KUKA KRL program: EPS_2_251806_MH42A_A_20260213065135.src

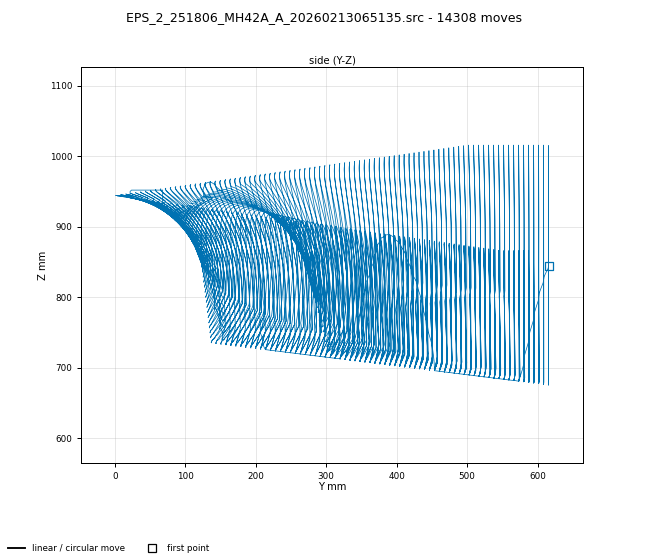
[picture p0: tool path of EPS_2_251806_MH42A_A_20260213065135.src, 14308 of 14310 moves have a stored position in this frame; points joined in program order, loops and branches not executed]
&ACCESS RVP
&REL 4
&COMMENT QRS 19112012
&PARAM EDITMASK = *
DEF PART()
EXT BAS (BAS_COMMAND :IN,REAL :IN )
INT I
BAS (#INITMOV,0 )

;KUKA QRS Post kuka4.cps  Date:22-06-2017 !

File_ID=3014

QRS_PRE_INIT()

;Init var - Until changes are made in qrs_pre_init
Outlet_Square_prg=0
Inlet_1_Square_prg=0
Inlet_2_Square_prg=0
Inlet_3_Square_prg=0
Inlet_4_Square_prg=0
Inlet_5_Square_prg=0

Outlet_1={X 0.000, Y 502.870, Z 915.500, B 0.000, E1 0.000 }
Inlet_1={X 0.000, Y 532.850, Z 495.500, B 0.000, E1 90.000 }
Inlet_2={X 0.000, Y 548.530, Z 275.500, B 0.000, E1 180.000 }
Outlet_1_type=201
Inlet_1_type=201
Inlet_2_type=201
;QRS#1=Sidecore dimensions
;QRS#2=200-8" PVC SDR 35
;QRS#3=200-8" PVC SDR 35
;QRS#4=200-8" PVC SDR 35
;QRS#5=
;QRS#6=
;QRS#7=
;QRS#8=
;QRS#9=12-08 PSX
;QRS#10=12-08 PSX
;QRS#11=12-08 PSX
;QRS#12=
;QRS#13=
;QRS#14=
;QRS#15=
;QRS#16=1220x127x1295 4,25'
;QRS#17=EPS Height
;QRS#18=1016
;QRS#19=*
;QRS#20= UPDATED VERSION 22-06-2017
;QRS#21=*
Outlet_Square=0100
Inlet_1_Square=0100
Inlet_2_Square=0100
Inlet_3_Square=0
Inlet_4_Square=0
Inlet_5_Square=0
Mill_Square=1
Outlet_Square_Prg=204
Inlet_1_Square_prg=204
Inlet_2_Square_prg=204

QRS_INIT()

$ADVANCE=5

; T1
PTP {E1 173.422,E2 173.422}
PTP {X 0,Y 615.492,A -85,B 0,C 180,E1 173.422,E2 173.422,E3 0,E4 0,E5 0,E6 0}
QRS_SPEED_INIT()
LIN {X 0,Y 615.492,Z 844.24,A -85,B 0,C 180,E1 173.422,E2 173.422,E3 0,E4 0,E5 0,E6 0} C_VEL
LIN {X 0,Y 615.497,Z 836.536,A -85,B 0,C 180,E1 172.455,E2 172.455} C_VEL
LIN {X 0,Y 615.498,Z 826.758,A -85,B 0,C 180,E1 171.463,E2 171.463} C_VEL
LIN {X 0,Y 615.497,Z 816.492,A -85,B 0,C 180,E1 170.636,E2 170.636} C_VEL
LIN {X 0,Y 615.468,Z 804.932,A -85,B 0,C 180,E1 169.888,E2 169.888} C_VEL
LIN {X 0,Y 615.49,Z 793.084,A -85,B 0,C 180,E1 169.293,E2 169.293} C_VEL
LIN {X 0,Y 615.491,Z 780.156,A -85,B 0,C 180,E1 168.807,E2 168.807} C_VEL
LIN {X 0,Y 615.484,Z 767.556,A -85,B 0,C 180,E1 168.473,E2 168.473} C_VEL
LIN {X 0,Y 615.469,Z 754.433,A -85,B 0,C 180,E1 168.264,E2 168.264} C_VEL
LIN {X 0,Y 615.494,Z 675.805,A -85,B 0,C 180,E1 167.344,E2 167.344} C_VEL
LIN {X 0,Y 615.486,Z 675.687,A -85,B 0,C 180,E1 164.774,E2 164.774} C_VEL
LIN {X 0,Y 615.473,Z 675.686,A -85,B 0,C 180,E1 162.043,E2 162.043} C_VEL
LIN {X 0,Y 615.491,Z 675.701,A -85,B 0,C 180,E1 159.269,E2 159.269} C_VEL
LIN {X 0,Y 615.483,Z 675.683,A -85,B 0,C 180,E1 156.443,E2 156.443} C_VEL
LIN {X 0,Y 615.479,Z 675.691,A -85,B 0,C 180,E1 153.555,E2 153.555} C_VEL
LIN {X 0,Y 615.487,Z 675.696,A -85,B 0,C 180,E1 151.342,E2 151.342} C_VEL
LIN {X 0,Y 615.478,Z 675.697,A -85,B 0,C 180,E1 148.917,E2 148.917} C_VEL
LIN {X 0,Y 615.465,Z 675.69,A -85,B 0,C 180,E1 146.471,E2 146.471} C_VEL
LIN {X 0,Y 615.468,Z 675.686,A -85,B 0,C 180,E1 144.171,E2 144.171} C_VEL
LIN {X 0,Y 615.479,Z 675.683,A -85,B 0,C 180,E1 141.931,E2 141.931} C_VEL
LIN {X 0,Y 615.486,Z 675.699,A -85,B 0,C 180,E1 138.908,E2 138.908} C_VEL
LIN {X 0,Y 615.474,Z 675.697,A -85,B 0,C 180,E1 136.754,E2 136.754} C_VEL
LIN {X 0,Y 615.447,Z 675.692,A -85,B 0,C 180,E1 134.155,E2 134.155} C_VEL
LIN {X 0,Y 615.487,Z 675.685,A -85,B 0,C 180,E1 131.476,E2 131.476} C_VEL
LIN {X 0,Y 615.493,Z 675.701,A -85,B 0,C 180,E1 128.906,E2 128.906} C_VEL
LIN {X 0,Y 615.45,Z 675.697,A -85,B 0,C 180,E1 126.43,E2 126.43} C_VEL
LIN {X 0,Y 615.431,Z 675.695,A -85,B 0,C 180,E1 124.028,E2 124.028} C_VEL
LIN {X 0,Y 615.432,Z 675.694,A -85,B 0,C 180,E1 121.691,E2 121.691} C_VEL
LIN {X 0,Y 615.443,Z 675.694,A -85,B 0,C 180,E1 119.411,E2 119.411} C_VEL
LIN {X 0,Y 615.456,Z 675.699,A -85,B 0,C 180,E1 116.448,E2 116.448} C_VEL
LIN {X 0,Y 615.415,Z 675.7,A -85,B 0,C 180,E1 113.992,E2 113.992} C_VEL
LIN {X 0,Y 615.425,Z 675.7,A -85,B 0,C 180,E1 112.142,E2 112.142} C_VEL
LIN {X 0,Y 615.418,Z 675.7,A -85,B 0,C 180,E1 110.038,E2 110.038} C_VEL
LIN {X 0,Y 615.418,Z 675.699,A -85,B 0,C 180,E1 107.962,E2 107.962} C_VEL
LIN {X 0,Y 615.422,Z 675.698,A -85,B 0,C 180,E1 105.91,E2 105.91} C_VEL
LIN {X 0,Y 615.427,Z 675.697,A -85,B 0,C 180,E1 103.879,E2 103.879} C_VEL
LIN {X 0,Y 615.489,Z 675.702,A -85,B 0,C 180,E1 102.576,E2 102.576} C_VEL
LIN {X 0,Y 615.42,Z 762.61,A -85,B 0,C 180,E1 101.532,E2 101.532} C_VEL
LIN {X 0,Y 615.425,Z 775.619,A -85,B 0,C 180,E1 101.24,E2 101.24} C_VEL
LIN {X 0,Y 615.46,Z 788.009,A -85,B 0,C 180,E1 100.828,E2 100.828} C_VEL
LIN {X 0,Y 615.489,Z 800.126,A -85,B 0,C 180,E1 100.281,E2 100.281} C_VEL
LIN {X 0,Y 615.483,Z 811.521,A -85,B 0,C 180,E1 99.617,E2 99.617} C_VEL
LIN {X 0,Y 615.498,Z 821.775,A -85,B 0,C 180,E1 98.871,E2 98.871} C_VEL
LIN {X 0,Y 615.498,Z 830.882,A -85,B 0,C 180,E1 98.044,E2 98.044} C_VEL
LIN {X 0,Y 615.497,Z 838.565,A -85,B 0,C 180,E1 97.219,E2 97.219} C_VEL
LIN {X 0,Y 615.497,Z 845.984,A -85,B 0,C 180,E1 96.231,E2 96.231} C_VEL
LIN {X 0,Y 615.497,Z 851.936,A -85,B 0,C 180,E1 95.245,E2 95.245} C_VEL
LIN {X 0,Y 615.493,Z 856.64,A -85,B 0,C 180,E1 94.26,E2 94.26} C_VEL
LIN {X 0,Y 615.494,Z 860.241,A -85,B 0,C 180,E1 93.277,E2 93.277} C_VEL
LIN {X 0,Y 615.496,Z 862.103,A -85,B 0,C 180,E1 92.622,E2 92.622} C_VEL
LIN {X 0,Y 615.497,Z 863.526,A -85,B 0,C 180,E1 91.967,E2 91.967} C_VEL
LIN {X 0,Y 615.496,Z 865.138,A -85,B 0,C 180,E1 90.659,E2 90.659} C_VEL
LIN {X 0,Y 615.495,Z 865.383,A -85,B 0,C 180,E1 90.004,E2 90.004} C_VEL
LIN {X 0,Y 615.495,Z 865.209,A -85,B 0,C 180,E1 89.35,E2 89.35} C_VEL
LIN {X 0,Y 615.497,Z 863.69,A -85,B 0,C 180,E1 88.041,E2 88.041} C_VEL
LIN {X 0,Y 615.498,Z 862.352,A -85,B 0,C 180,E1 87.387,E2 87.387} C_VEL
LIN {X 0,Y 615.496,Z 859.509,A -85,B 0,C 180,E1 86.404,E2 86.404} C_VEL
LIN {X 0,Y 615.499,Z 855.654,A -85,B 0,C 180,E1 85.42,E2 85.42} C_VEL
LIN {X 0,Y 615.498,Z 850.677,A -85,B 0,C 180,E1 84.435,E2 84.435} C_VEL
LIN {X 0,Y 615.488,Z 844.256,A -85,B 0,C 180,E1 83.424,E2 83.424} C_VEL
LIN {X 0,Y 615.497,Z 836.581,A -85,B 0,C 180,E1 82.46,E2 82.46} C_VEL
LIN {X 0,Y 615.498,Z 826.813,A -85,B 0,C 180,E1 81.469,E2 81.469} C_VEL
LIN {X 0,Y 615.497,Z 816.563,A -85,B 0,C 180,E1 80.641,E2 80.641} C_VEL
LIN {X 0,Y 615.486,Z 805.017,A -85,B 0,C 180,E1 79.894,E2 79.894} C_VEL
LIN {X 0,Y 615.485,Z 793.267,A -85,B 0,C 180,E1 79.301,E2 79.301} C_VEL
LIN {X 0,Y 615.438,Z 780.329,A -85,B 0,C 180,E1 78.811,E2 78.811} C_VEL
LIN {X 0,Y 615.427,Z 767.799,A -85,B 0,C 180,E1 78.477,E2 78.477} C_VEL
LIN {X 0,Y 615.431,Z 754.903,A -85,B 0,C 180,E1 78.269,E2 78.269} C_VEL
LIN {X 0,Y 615.491,Z 675.701,A -85,B 0,C 180,E1 77.329,E2 77.329} C_VEL
LIN {X 0,Y 615.444,Z 675.697,A -85,B 0,C 180,E1 74.778,E2 74.778} C_VEL
LIN {X 0,Y 615.445,Z 675.698,A -85,B 0,C 180,E1 72.734,E2 72.734} C_VEL
LIN {X 0,Y 615.441,Z 675.698,A -85,B 0,C 180,E1 70.667,E2 70.667} C_VEL
LIN {X 0,Y 615.441,Z 675.698,A -85,B 0,C 180,E1 68.573,E2 68.573} C_VEL
LIN {X 0,Y 615.435,Z 675.698,A -85,B 0,C 180,E1 66.448,E2 66.448} C_VEL
LIN {X 0,Y 615.429,Z 675.697,A -85,B 0,C 180,E1 64.288,E2 64.288} C_VEL
LIN {X 0,Y 615.424,Z 675.696,A -85,B 0,C 180,E1 62.089,E2 62.089} C_VEL
LIN {X 0,Y 615.422,Z 675.696,A -85,B 0,C 180,E1 59.844,E2 59.844} C_VEL
LIN {X 0,Y 615.428,Z 675.695,A -85,B 0,C 180,E1 57.547,E2 57.547} C_VEL
LIN {X 0,Y 615.45,Z 675.694,A -85,B 0,C 180,E1 55.191,E2 55.191} C_VEL
LIN {X 0,Y 615.49,Z 675.694,A -85,B 0,C 180,E1 52.766,E2 52.766} C_VEL
LIN {X 0,Y 615.43,Z 675.698,A -85,B 0,C 180,E1 49.918,E2 49.918} C_VEL
LIN {X 0,Y 615.42,Z 675.697,A -85,B 0,C 180,E1 47.651,E2 47.651} C_VEL
LIN {X 0,Y 615.439,Z 675.695,A -85,B 0,C 180,E1 44.937,E2 44.937} C_VEL
LIN {X 0,Y 615.474,Z 675.7,A -85,B 0,C 180,E1 42.09,E2 42.09} C_VEL
LIN {X 0,Y 615.44,Z 675.699,A -85,B 0,C 180,E1 39.754,E2 39.754} C_VEL
LIN {X 0,Y 615.411,Z 675.698,A -85,B 0,C 180,E1 37.248,E2 37.248} C_VEL
LIN {X 0,Y 615.428,Z 675.696,A -85,B 0,C 180,E1 34.706,E2 34.706} C_VEL
LIN {X 0,Y 615.458,Z 675.696,A -85,B 0,C 180,E1 32.341,E2 32.341} C_VEL
LIN {X 0,Y 615.434,Z 675.699,A -85,B 0,C 180,E1 29.409,E2 29.409} C_VEL
LIN {X 0,Y 615.414,Z 675.698,A -85,B 0,C 180,E1 27.049,E2 27.049} C_VEL
LIN {X 0,Y 615.414,Z 675.699,A -85,B 0,C 180,E1 24.995,E2 24.995} C_VEL
LIN {X 0,Y 615.407,Z 675.699,A -85,B 0,C 180,E1 22.848,E2 22.848} C_VEL
LIN {X 0,Y 615.409,Z 675.698,A -85,B 0,C 180,E1 20.56,E2 20.56} C_VEL
LIN {X 0,Y 615.444,Z 675.698,A -85,B 0,C 180,E1 17.958,E2 17.958} C_VEL
LIN {X 0,Y 615.462,Z 675.7,A -85,B 0,C 180,E1 15.227,E2 15.227} C_VEL
LIN {X 0,Y 615.407,Z 675.699,A -85,B 0,C 180,E1 12.532,E2 12.532} C_VEL
LIN {X 0,Y 615.408,Z 675.699,A -85,B 0,C 180,E1 10.528,E2 10.528} C_VEL
LIN {X 0,Y 615.411,Z 675.7,A -85,B 0,C 180,E1 8.538,E2 8.538} C_VEL
LIN {X 0,Y 615.415,Z 675.7,A -85,B 0,C 180,E1 6.558,E2 6.558} C_VEL
LIN {X 0,Y 615.422,Z 675.7,A -85,B 0,C 180,E1 4.585,E2 4.585} C_VEL
LIN {X 0,Y 615.43,Z 675.7,A -85,B 0,C 180,E1 2.618,E2 2.618} C_VEL
LIN {X 0,Y 615.401,Z 675.7,A -85,B 0,C 180,E1 0,E2 0} C_VEL
LIN {X 0,Y 615.431,Z 675.7,A -85,B 0,C 180,E1 -2.618,E2 -2.618} C_VEL
LIN {X 0,Y 615.479,Z 675.701,A -85,B 0,C 180,E1 -5.241,E2 -5.241} C_VEL
LIN {X 0,Y 615.418,Z 675.699,A -85,B 0,C 180,E1 -7.877,E2 -7.877} C_VEL
LIN {X 0,Y 615.425,Z 675.699,A -85,B 0,C 180,E1 -9.863,E2 -9.863} C_VEL
LIN {X 0,Y 615.431,Z 675.699,A -85,B 0,C 180,E1 -11.862,E2 -11.862} C_VEL
LIN {X 0,Y 615.431,Z 675.698,A -85,B 0,C 180,E1 -13.945,E2 -13.945} C_VEL
LIN {X 0,Y 615.408,Z 675.699,A -85,B 0,C 180,E1 -16.435,E2 -16.435} C_VEL
LIN {X 0,Y 615.408,Z 675.699,A -85,B 0,C 180,E1 -18.649,E2 -18.649} C_VEL
LIN {X 0,Y 615.466,Z 675.7,A -85,B 0,C 180,E1 -21.433,E2 -21.433} C_VEL
LIN {X 0,Y 615.434,Z 675.697,A -85,B 0,C 180,E1 -24.274,E2 -24.274} C_VEL
LIN {X 0,Y 615.425,Z 675.697,A -85,B 0,C 180,E1 -26.447,E2 -26.447} C_VEL
LIN {X 0,Y 615.417,Z 675.697,A -85,B 0,C 180,E1 -28.662,E2 -28.662} C_VEL
LIN {X 0,Y 615.412,Z 675.698,A -85,B 0,C 180,E1 -30.924,E2 -30.924} C_VEL
LIN {X 0,Y 615.436,Z 675.699,A -85,B 0,C 180,E1 -33.541,E2 -33.541} C_VEL
LIN {X 0,Y 615.466,Z 675.695,A -85,B 0,C 180,E1 -36.426,E2 -36.426} C_VEL
LIN {X 0,Y 615.425,Z 675.696,A -85,B 0,C 180,E1 -38.909,E2 -38.909} C_VEL
LIN {X 0,Y 615.419,Z 675.696,A -85,B 0,C 180,E1 -41.098,E2 -41.098} C_VEL
LIN {X 0,Y 615.418,Z 675.696,A -85,B 0,C 180,E1 -43.251,E2 -43.251} C_VEL
LIN {X 0,Y 615.434,Z 675.698,A -85,B 0,C 180,E1 -45.856,E2 -45.856} C_VEL
LIN {X 0,Y 615.497,Z 675.697,A -85,B 0,C 180,E1 -48.536,E2 -48.536} C_VEL
LIN {X 0,Y 615.442,Z 675.695,A -85,B 0,C 180,E1 -51.101,E2 -51.101} C_VEL
LIN {X 0,Y 615.421,Z 675.696,A -85,B 0,C 180,E1 -53.579,E2 -53.579} C_VEL
LIN {X 0,Y 615.469,Z 675.699,A -85,B 0,C 180,E1 -56.469,E2 -56.469} C_VEL
LIN {X 0,Y 615.475,Z 675.693,A -85,B 0,C 180,E1 -59.087,E2 -59.087} C_VEL
LIN {X 0,Y 615.437,Z 675.694,A -85,B 0,C 180,E1 -61.559,E2 -61.559} C_VEL
LIN {X 0,Y 615.423,Z 675.695,A -85,B 0,C 180,E1 -63.924,E2 -63.924} C_VEL
LIN {X 0,Y 615.422,Z 675.729,A -85,B 0,C 180,E1 -64.061,E2 -64.061} C_VEL
LIN {X 0,Y 615.468,Z 698.001,A -85,B 0,C 180,E1 -66.449,E2 -66.449} C_VEL
LIN {X 0,Y 615.49,Z 724.895,A -85,B 0,C 180,E1 -69.276,E2 -69.276} C_VEL
LIN {X 0,Y 615.484,Z 753.464,A -85,B 0,C 180,E1 -72.221,E2 -72.221} C_VEL
LIN {X 0,Y 615.437,Z 778.642,A -85,B 0,C 180,E1 -74.778,E2 -74.778} C_VEL
LIN {X 0,Y 615.451,Z 801.694,A -85,B 0,C 180,E1 -77.097,E2 -77.097} C_VEL
LIN {X 0,Y 615.434,Z 912.129,A -85,B 0,C 180,E1 -78.415,E2 -78.415} C_VEL
LIN {X 0,Y 615.441,Z 924.542,A -85,B 0,C 180,E1 -78.686,E2 -78.686} C_VEL
LIN {X 0,Y 615.479,Z 937.74,A -85,B 0,C 180,E1 -79.117,E2 -79.117} C_VEL
LIN {X 0,Y 615.492,Z 949.575,A -85,B 0,C 180,E1 -79.645,E2 -79.645} C_VEL
LIN {X 0,Y 615.483,Z 961.074,A -85,B 0,C 180,E1 -80.309,E2 -80.309} C_VEL
LIN {X 0,Y 615.499,Z 971.405,A -85,B 0,C 180,E1 -81.055,E2 -81.055} C_VEL
LIN {X 0,Y 615.497,Z 979.742,A -85,B 0,C 180,E1 -81.799,E2 -81.799} C_VEL
LIN {X 0,Y 615.497,Z 987.648,A -85,B 0,C 180,E1 -82.624,E2 -82.624} C_VEL
LIN {X 0,Y 615.491,Z 995.236,A -85,B 0,C 180,E1 -83.613,E2 -83.613} C_VEL
LIN {X 0,Y 615.498,Z 1002.23,A -85,B 0,C 180,E1 -84.764,E2 -84.764} C_VEL
LIN {X 0,Y 615.493,Z 1006.871,A -85,B 0,C 180,E1 -85.748,E2 -85.748} C_VEL
LIN {X 0,Y 615.494,Z 1010.413,A -85,B 0,C 180,E1 -86.732,E2 -86.732} C_VEL
LIN {X 0,Y 615.497,Z 1012.244,A -85,B 0,C 180,E1 -87.387,E2 -87.387} C_VEL
LIN {X 0,Y 615.497,Z 1013.616,A -85,B 0,C 180,E1 -88.041,E2 -88.041} C_VEL
LIN {X 0,Y 615.496,Z 1015.177,A -85,B 0,C 180,E1 -89.35,E2 -89.35} C_VEL
LIN {X 0,Y 615.494,Z 1015.389,A -85,B 0,C 180,E1 -90.004,E2 -90.004} C_VEL
LIN {X 0,Y 615.495,Z 1014.575,A -85,B 0,C 180,E1 -91.313,E2 -91.313} C_VEL
LIN {X 0,Y 615.497,Z 1013.601,A -85,B 0,C 180,E1 -91.967,E2 -91.967} C_VEL
LIN {X 0,Y 615.497,Z 1012.222,A -85,B 0,C 180,E1 -92.622,E2 -92.622} C_VEL
LIN {X 0,Y 615.495,Z 1009.336,A -85,B 0,C 180,E1 -93.605,E2 -93.605} C_VEL
LIN {X 0,Y 615.497,Z 1005.424,A -85,B 0,C 180,E1 -94.589,E2 -94.589} C_VEL
LIN {X 0,Y 615.499,Z 1000.383,A -85,B 0,C 180,E1 -95.574,E2 -95.574} C_VEL
LIN {X 0,Y 615.49,Z 993.913,A -85,B 0,C 180,E1 -96.578,E2 -96.578} C_VEL
LIN {X 0,Y 615.497,Z 986.099,A -85,B 0,C 180,E1 -97.549,E2 -97.549} C_VEL
LIN {X 0,Y 615.498,Z 976.214,A -85,B 0,C 180,E1 -98.54,E2 -98.54} C_VEL
LIN {X 0,Y 615.495,Z 965.813,A -85,B 0,C 180,E1 -99.368,E2 -99.368} C_VEL
LIN {X 0,Y 615.482,Z 955.513,A -85,B 0,C 180,E1 -100.032,E2 -100.032} C_VEL
LIN {X 0,Y 615.494,Z 944.086,A -85,B 0,C 180,E1 -100.618,E2 -100.618} C_VEL
LIN {X 0,Y 615.457,Z 932.311,A -85,B 0,C 180,E1 -101.079,E2 -101.079} C_VEL
LIN {X 0,Y 615.436,Z 919.092,A -85,B 0,C 180,E1 -101.448,E2 -101.448} C_VEL
LIN {X 0,Y 615.435,Z 905.652,A -85,B 0,C 180,E1 -101.677,E2 -101.677} C_VEL
LIN {X 0,Y 615.45,Z 801.605,A -85,B 0,C 180,E1 -102.912,E2 -102.912} C_VEL
LIN {X 0,Y 615.438,Z 776.876,A -85,B 0,C 180,E1 -105.4,E2 -105.4} C_VEL
LIN {X 0,Y 615.497,Z 751.695,A -85,B 0,C 180,E1 -107.96,E2 -107.96} C_VEL
LIN {X 0,Y 615.49,Z 724.806,A -85,B 0,C 180,E1 -110.734,E2 -110.734} C_VEL
LIN {X 0,Y 615.467,Z 697.911,A -85,B 0,C 180,E1 -113.56,E2 -113.56} C_VEL
LIN {X 0,Y 615.422,Z 675.85,A -85,B 0,C 180,E1 -115.926,E2 -115.926} C_VEL
LIN {X 0,Y 615.417,Z 675.698,A -85,B 0,C 180,E1 -117.921,E2 -117.921} C_VEL
LIN {X 0,Y 615.414,Z 675.698,A -85,B 0,C 180,E1 -120.167,E2 -120.167} C_VEL
LIN {X 0,Y 615.42,Z 675.699,A -85,B 0,C 180,E1 -122.464,E2 -122.464} C_VEL
LIN {X 0,Y 615.449,Z 675.7,A -85,B 0,C 180,E1 -124.82,E2 -124.82} C_VEL
LIN {X 0,Y 615.489,Z 675.699,A -85,B 0,C 180,E1 -127.244,E2 -127.244} C_VEL
LIN {X 0,Y 615.441,Z 675.696,A -85,B 0,C 180,E1 -129.756,E2 -129.756} C_VEL
LIN {X 0,Y 615.427,Z 675.695,A -85,B 0,C 180,E1 -132.074,E2 -132.074} C_VEL
LIN {X 0,Y 615.43,Z 675.695,A -85,B 0,C 180,E1 -134.157,E2 -134.157} C_VEL
LIN {X 0,Y 615.464,Z 675.698,A -85,B 0,C 180,E1 -136.957,E2 -136.957} C_VEL
LIN {X 0,Y 615.468,Z 675.688,A -85,B 0,C 180,E1 -139.915,E2 -139.915} C_VEL
LIN {X 0,Y 615.451,Z 675.695,A -85,B 0,C 180,E1 -142.755,E2 -142.755} C_VEL
LIN {X 0,Y 615.491,Z 675.701,A -85,B 0,C 180,E1 -145.301,E2 -145.301} C_VEL
LIN {X 0,Y 615.464,Z 675.687,A -85,B 0,C 180,E1 -148.313,E2 -148.313} C_VEL
LIN {X 0,Y 615.46,Z 675.689,A -85,B 0,C 180,E1 -150.592,E2 -150.592} C_VEL
LIN {X 0,Y 615.469,Z 675.694,A -85,B 0,C 180,E1 -152.96,E2 -152.96} C_VEL
LIN {X 0,Y 615.483,Z 675.691,A -85,B 0,C 180,E1 -155.728,E2 -155.728} C_VEL
LIN {X 0,Y 615.478,Z 675.684,A -85,B 0,C 180,E1 -158.568,E2 -158.568} C_VEL
LIN {X 0,Y 615.492,Z 675.702,A -85,B 0,C 180,E1 -161.396,E2 -161.396} C_VEL
LIN {X 0,Y 615.475,Z 675.686,A -85,B 0,C 180,E1 -164.094,E2 -164.094} C_VEL
LIN {X 0,Y 615.486,Z 675.685,A -85,B 0,C 180,E1 -166.799,E2 -166.799} C_VEL
LIN {X 0,Y 615.491,Z 675.702,A -85,B 0,C 180,E1 -167.428,E2 -167.428} C_VEL
LIN {X 0,Y 615.484,Z 761.644,A -85,B 0,C 180,E1 -168.452,E2 -168.452} C_VEL
LIN {X 0,Y 615.493,Z 774.222,A -85,B 0,C 180,E1 -168.724,E2 -168.724} C_VEL
LIN {X 0,Y 615.485,Z 786.478,A -85,B 0,C 180,E1 -169.116,E2 -169.116} C_VEL
LIN {X 0,Y 615.482,Z 798.567,A -85,B 0,C 180,E1 -169.639,E2 -169.639} C_VEL
LIN {X 0,Y 615.474,Z 810.307,A -85,B 0,C 180,E1 -170.304,E2 -170.304} C_VEL
LIN {X 0,Y 615.499,Z 820.768,A -85,B 0,C 180,E1 -171.05,E2 -171.05} C_VEL
LIN {X 0,Y 615.498,Z 829.231,A -85,B 0,C 180,E1 -171.794,E2 -171.794} C_VEL
LIN {X 0,Y 615.497,Z 837.209,A -85,B 0,C 180,E1 -172.62,E2 -172.62} C_VEL
LIN {X 0,Y 615.491,Z 844.9,A -85,B 0,C 180,E1 -173.608,E2 -173.608} C_VEL
LIN {X 0,Y 615.497,Z 851.958,A -85,B 0,C 180,E1 -174.759,E2 -174.759} C_VEL
LIN {X 0,Y 615.493,Z 856.658,A -85,B 0,C 180,E1 -175.744,E2 -175.744} C_VEL
LIN {X 0,Y 615.496,Z 860.254,A -85,B 0,C 180,E1 -176.727,E2 -176.727} C_VEL
LIN {X 0,Y 615.496,Z 862.115,A -85,B 0,C 180,E1 -177.382,E2 -177.382} C_VEL
LIN {X 0,Y 615.497,Z 863.534,A -85,B 0,C 180,E1 -178.037,E2 -178.037} C_VEL
LIN {X 0,Y 615.496,Z 865.142,A -85,B 0,C 180,E1 -179.346,E2 -179.346} C_VEL
LIN {X 0,Y 615.494,Z 865.384,A -85,B 0,C 180,E1 -180,E2 -180} C_VEL
LIN {X 0,Y 615.495,Z 865.206,A -85,B 0,C 180,E1 -180.654,E2 -180.654} C_VEL
LIN {X 0,Y 615.496,Z 863.683,A -85,B 0,C 180,E1 -181.963,E2 -181.963} C_VEL
LIN {X 0,Y 615.498,Z 862.341,A -85,B 0,C 180,E1 -182.618,E2 -182.618} C_VEL
LIN {X 0,Y 615.496,Z 859.494,A -85,B 0,C 180,E1 -183.601,E2 -183.601} C_VEL
LIN {X 0,Y 615.498,Z 855.634,A -85,B 0,C 180,E1 -184.585,E2 -184.585} C_VEL
LIN {X 0,Y 615.498,Z 850.651,A -85,B 0,C 180,E1 -185.57,E2 -185.57} C_VEL
LIN {X 0,Y 615.492,Z 844.24,A -85,B 0,C 180,E1 -186.578,E2 -186.578} C_VEL
LIN {X 0,Y 614.826,Z 841.059,A -85,B 0,C 180,E1 -187.027,E2 -187.027} C_VEL
LIN {X 0,Y 611.988,Z 835.485,A -85,B 0,C 180,E1 -187.745,E2 -187.745} C_VEL
LIN {X 0,Y 609.138,Z 829.212,A -85,B 0,C 180,E1 -188.426,E2 -188.426} C_VEL
LIN {X 0,Y 608.477,Z 824.972,A -85,B 0,C 180,E1 -188.816,E2 -188.816} C_VEL
LIN {X 0,Y 608.486,Z 814.391,A -85,B 0,C 180,E1 -189.641,E2 -189.641} C_VEL
LIN {X 0,Y 608.476,Z 803.599,A -85,B 0,C 180,E1 -190.313,E2 -190.313} C_VEL
LIN {X 0,Y 608.53,Z 791.933,A -85,B 0,C 180,E1 -190.885,E2 -190.885} C_VEL
LIN {X 0,Y 608.525,Z 778.959,A -85,B 0,C 180,E1 -191.365,E2 -191.365} C_VEL
LIN {X 0,Y 608.536,Z 766.652,A -85,B 0,C 180,E1 -191.681,E2 -191.681} C_VEL
LIN {X 0,Y 608.53,Z 752.744,A -85,B 0,C 180,E1 -191.893,E2 -191.893} C_VEL
LIN {X 0,Y 608.458,Z 676.695,A -85,B 0,C 180,E1 -192.805,E2 -192.805} C_VEL
LIN {X 0,Y 608.467,Z 676.686,A -85,B 0,C 180,E1 -195.406,E2 -195.406} C_VEL
LIN {X 0,Y 608.44,Z 676.691,A -85,B 0,C 180,E1 -198.172,E2 -198.172} C_VEL
LIN {X 0,Y 608.458,Z 676.693,A -85,B 0,C 180,E1 -200.982,E2 -200.982} C_VEL
LIN {X 0,Y 608.464,Z 676.685,A -85,B 0,C 180,E1 -203.845,E2 -203.845} C_VEL
LIN {X 0,Y 608.444,Z 676.688,A -85,B 0,C 180,E1 -206.036,E2 -206.036} C_VEL
LIN {X 0,Y 608.473,Z 676.691,A -85,B 0,C 180,E1 -208.618,E2 -208.618} C_VEL
LIN {X 0,Y 608.448,Z 676.691,A -85,B 0,C 180,E1 -211.318,E2 -211.318} C_VEL
LIN {X 0,Y 608.456,Z 676.687,A -85,B 0,C 180,E1 -213.731,E2 -213.731} C_VEL
LIN {X 0,Y 608.451,Z 676.687,A -85,B 0,C 180,E1 -216.092,E2 -216.092} C_VEL
LIN {X 0,Y 608.446,Z 676.692,A -85,B 0,C 180,E1 -218.59,E2 -218.59} C_VEL
LIN {X 0,Y 608.448,Z 676.692,A -85,B 0,C 180,E1 -221.339,E2 -221.339} C_VEL
LIN {X 0,Y 608.447,Z 676.688,A -85,B 0,C 180,E1 -223.872,E2 -223.872} C_VEL
LIN {X 0,Y 608.481,Z 676.688,A -85,B 0,C 180,E1 -226.69,E2 -226.69} C_VEL
LIN {X 0,Y 608.463,Z 676.692,A -85,B 0,C 180,E1 -228.822,E2 -228.822} C_VEL
LIN {X 0,Y 608.428,Z 676.696,A -85,B 0,C 180,E1 -231.406,E2 -231.406} C_VEL
LIN {X 0,Y 608.456,Z 676.697,A -85,B 0,C 180,E1 -233.083,E2 -233.083} C_VEL
LIN {X 0,Y 608.452,Z 676.692,A -85,B 0,C 180,E1 -235.527,E2 -235.527} C_VEL
LIN {X 0,Y 608.424,Z 676.691,A -85,B 0,C 180,E1 -237.9,E2 -237.9} C_VEL
LIN {X 0,Y 608.412,Z 676.692,A -85,B 0,C 180,E1 -240.215,E2 -240.215} C_VEL
LIN {X 0,Y 608.442,Z 676.691,A -85,B 0,C 180,E1 -242.8,E2 -242.8} C_VEL
LIN {X 0,Y 608.401,Z 676.695,A -85,B 0,C 180,E1 -245.864,E2 -245.864} C_VEL
LIN {X 0,Y 608.381,Z 676.696,A -85,B 0,C 180,E1 -248.302,E2 -248.302} C_VEL
LIN {X 0,Y 608.39,Z 676.695,A -85,B 0,C 180,E1 -250.424,E2 -250.424} C_VEL
LIN {X 0,Y 608.393,Z 676.694,A -85,B 0,C 180,E1 -252.518,E2 -252.518} C_VEL
LIN {X 0,Y 608.389,Z 676.695,A -85,B 0,C 180,E1 -254.588,E2 -254.588} C_VEL
LIN {X 0,Y 608.479,Z 676.872,A -85,B 0,C 180,E1 -257.298,E2 -257.298} C_VEL
LIN {X 0,Y 608.49,Z 762.745,A -85,B 0,C 180,E1 -258.335,E2 -258.335} C_VEL
LIN {X 0,Y 608.461,Z 776.507,A -85,B 0,C 180,E1 -258.651,E2 -258.651} C_VEL
LIN {X 0,Y 608.485,Z 787.939,A -85,B 0,C 180,E1 -259.038,E2 -259.038} C_VEL
LIN {X 0,Y 608.505,Z 800.289,A -85,B 0,C 180,E1 -259.6,E2 -259.6} C_VEL
LIN {X 0,Y 608.493,Z 811.722,A -85,B 0,C 180,E1 -260.271,E2 -260.271} C_VEL
LIN {X 0,Y 608.475,Z 822.026,A -85,B 0,C 180,E1 -261.026,E2 -261.026} C_VEL
LIN {X 0,Y 608.464,Z 831.203,A -85,B 0,C 180,E1 -261.862,E2 -261.862} C_VEL
LIN {X 0,Y 608.463,Z 838.934,A -85,B 0,C 180,E1 -262.697,E2 -262.697} C_VEL
LIN {X 0,Y 608.449,Z 846.41,A -85,B 0,C 180,E1 -263.696,E2 -263.696} C_VEL
LIN {X 0,Y 608.462,Z 852.413,A -85,B 0,C 180,E1 -264.694,E2 -264.694} C_VEL
LIN {X 0,Y 608.439,Z 857.161,A -85,B 0,C 180,E1 -265.69,E2 -265.69} C_VEL
LIN {X 0,Y 608.425,Z 860.799,A -85,B 0,C 180,E1 -266.685,E2 -266.685} C_VEL
LIN {X 0,Y 608.425,Z 862.679,A -85,B 0,C 180,E1 -267.348,E2 -267.348} C_VEL
LIN {X 0,Y 608.442,Z 864.119,A -85,B 0,C 180,E1 -268.01,E2 -268.01} C_VEL
LIN {X 0,Y 608.439,Z 865.749,A -85,B 0,C 180,E1 -269.334,E2 -269.334} C_VEL
LIN {X 0,Y 608.435,Z 865.994,A -85,B 0,C 180,E1 -269.996,E2 -269.996} C_VEL
LIN {X 0,Y 608.438,Z 865.818,A -85,B 0,C 180,E1 -270.657,E2 -270.657} C_VEL
LIN {X 0,Y 608.442,Z 864.284,A -85,B 0,C 180,E1 -271.981,E2 -271.981} C_VEL
LIN {X 0,Y 608.426,Z 862.929,A -85,B 0,C 180,E1 -272.644,E2 -272.644} C_VEL
LIN {X 0,Y 608.449,Z 860.057,A -85,B 0,C 180,E1 -273.638,E2 -273.638} C_VEL
LIN {X 0,Y 608.433,Z 856.164,A -85,B 0,C 180,E1 -274.633,E2 -274.633} C_VEL
LIN {X 0,Y 608.449,Z 851.139,A -85,B 0,C 180,E1 -275.63,E2 -275.63} C_VEL
LIN {X 0,Y 608.434,Z 844.828,A -85,B 0,C 180,E1 -276.628,E2 -276.628} C_VEL
LIN {X 0,Y 608.474,Z 836.917,A -85,B 0,C 180,E1 -277.628,E2 -277.628} C_VEL
LIN {X 0,Y 608.471,Z 827.084,A -85,B 0,C 180,E1 -278.631,E2 -278.631} C_VEL
LIN {X 0,Y 608.478,Z 816.787,A -85,B 0,C 180,E1 -279.468,E2 -279.468} C_VEL
LIN {X 0,Y 608.483,Z 805.19,A -85,B 0,C 180,E1 -280.224,E2 -280.224} C_VEL
LIN {X 0,Y 608.5,Z 793.1,A -85,B 0,C 180,E1 -280.836,E2 -280.836} C_VEL
LIN {X 0,Y 608.486,Z 780.417,A -85,B 0,C 180,E1 -281.318,E2 -281.318} C_VEL
LIN {X 0,Y 608.491,Z 767.871,A -85,B 0,C 180,E1 -281.656,E2 -281.656} C_VEL
LIN {X 0,Y 608.5,Z 754.992,A -85,B 0,C 180,E1 -281.867,E2 -281.867} C_VEL
LIN {X 0,Y 608.471,Z 676.694,A -85,B 0,C 180,E1 -282.799,E2 -282.799} C_VEL
LIN {X 0,Y 608.428,Z 676.691,A -85,B 0,C 180,E1 -285.401,E2 -285.401} C_VEL
LIN {X 0,Y 608.41,Z 676.693,A -85,B 0,C 180,E1 -287.472,E2 -287.472} C_VEL
LIN {X 0,Y 608.406,Z 676.694,A -85,B 0,C 180,E1 -289.566,E2 -289.566} C_VEL
LIN {X 0,Y 608.422,Z 676.691,A -85,B 0,C 180,E1 -291.687,E2 -291.687} C_VEL
LIN {X 0,Y 608.424,Z 676.69,A -85,B 0,C 180,E1 -294.14,E2 -294.14} C_VEL
LIN {X 0,Y 608.475,Z 676.694,A -85,B 0,C 180,E1 -297.206,E2 -297.206} C_VEL
LIN {X 0,Y 608.395,Z 676.694,A -85,B 0,C 180,E1 -299.959,E2 -299.959} C_VEL
LIN {X 0,Y 608.412,Z 676.692,A -85,B 0,C 180,E1 -302.09,E2 -302.09} C_VEL
LIN {X 0,Y 608.442,Z 676.691,A -85,B 0,C 180,E1 -304.904,E2 -304.904} C_VEL
LIN {X 0,Y 608.432,Z 676.695,A -85,B 0,C 180,E1 -307.74,E2 -307.74} C_VEL
LIN {X 0,Y 608.391,Z 676.695,A -85,B 0,C 180,E1 -310.322,E2 -310.322} C_VEL
LIN {X 0,Y 608.392,Z 676.695,A -85,B 0,C 180,E1 -312.327,E2 -312.327} C_VEL
LIN {X 0,Y 608.398,Z 676.693,A -85,B 0,C 180,E1 -314.791,E2 -314.791} C_VEL
LIN {X 0,Y 608.487,Z 676.692,A -85,B 0,C 180,E1 -317.652,E2 -317.652} C_VEL
LIN {X 0,Y 608.417,Z 676.691,A -85,B 0,C 180,E1 -320.556,E2 -320.556} C_VEL
LIN {X 0,Y 608.389,Z 676.695,A -85,B 0,C 180,E1 -323.08,E2 -323.08} C_VEL
LIN {X 0,Y 608.43,Z 676.693,A -85,B 0,C 180,E1 -325.528,E2 -325.528} C_VEL
LIN {X 0,Y 608.436,Z 676.697,A -85,B 0,C 180,E1 -327.904,E2 -327.904} C_VEL
LIN {X 0,Y 608.464,Z 676.694,A -85,B 0,C 180,E1 -330.22,E2 -330.22} C_VEL
LIN {X 0,Y 608.382,Z 676.695,A -85,B 0,C 180,E1 -333.222,E2 -333.222} C_VEL
LIN {X 0,Y 608.406,Z 676.696,A -85,B 0,C 180,E1 -334.697,E2 -334.697} C_VEL
LIN {X 0,Y 608.395,Z 676.696,A -85,B 0,C 180,E1 -336.874,E2 -336.874} C_VEL
LIN {X 0,Y 608.39,Z 676.694,A -85,B 0,C 180,E1 -339.318,E2 -339.318} C_VEL
LIN {X 0,Y 608.394,Z 676.695,A -85,B 0,C 180,E1 -341.826,E2 -341.826} C_VEL
LIN {X 0,Y 608.437,Z 676.699,A -85,B 0,C 180,E1 -344.593,E2 -344.593} C_VEL
LIN {X 0,Y 608.408,Z 676.693,A -85,B 0,C 180,E1 -347.322,E2 -347.322} C_VEL
LIN {X 0,Y 608.395,Z 676.695,A -85,B 0,C 180,E1 -349.349,E2 -349.349} C_VEL
LIN {X 0,Y 608.391,Z 676.696,A -85,B 0,C 180,E1 -351.363,E2 -351.363} C_VEL
LIN {X 0,Y 608.392,Z 676.696,A -85,B 0,C 180,E1 -353.366,E2 -353.366} C_VEL
LIN {X 0,Y 608.394,Z 676.696,A -85,B 0,C 180,E1 -355.362,E2 -355.362} C_VEL
LIN {X 0,Y 608.421,Z 676.694,A -85,B 0,C 180,E1 -357.352,E2 -357.352} C_VEL
LIN {X 0,Y 608.392,Z 676.694,A -85,B 0,C 180,E1 -360,E2 -360} C_VEL
LIN {X 0,Y 608.421,Z 676.694,A -85,B 0,C 180,E1 -362.648,E2 -362.648} C_VEL
LIN {X 0,Y 608.467,Z 676.693,A -85,B 0,C 180,E1 -365.302,E2 -365.302} C_VEL
LIN {X 0,Y 608.406,Z 676.693,A -85,B 0,C 180,E1 -367.968,E2 -367.968} C_VEL
LIN {X 0,Y 608.391,Z 676.695,A -85,B 0,C 180,E1 -369.978,E2 -369.978} C_VEL
LIN {X 0,Y 608.398,Z 676.695,A -85,B 0,C 180,E1 -372.001,E2 -372.001} C_VEL
LIN {X 0,Y 608.393,Z 676.695,A -85,B 0,C 180,E1 -374.039,E2 -374.039} C_VEL
LIN {X 0,Y 608.394,Z 676.694,A -85,B 0,C 180,E1 -376.534,E2 -376.534} C_VEL
LIN {X 0,Y 608.389,Z 676.695,A -85,B 0,C 180,E1 -378.872,E2 -378.872} C_VEL
LIN {X 0,Y 608.435,Z 676.699,A -85,B 0,C 180,E1 -381.693,E2 -381.693} C_VEL
LIN {X 0,Y 608.39,Z 676.694,A -85,B 0,C 180,E1 -384.574,E2 -384.574} C_VEL
LIN {X 0,Y 608.422,Z 676.697,A -85,B 0,C 180,E1 -386.037,E2 -386.037} C_VEL
LIN {X 0,Y 608.409,Z 676.692,A -85,B 0,C 180,E1 -389.023,E2 -389.023} C_VEL
LIN {X 0,Y 608.414,Z 676.693,A -85,B 0,C 180,E1 -391.32,E2 -391.32} C_VEL
LIN {X 0,Y 608.438,Z 676.695,A -85,B 0,C 180,E1 -393.744,E2 -393.744} C_VEL
LIN {X 0,Y 608.43,Z 676.701,A -85,B 0,C 180,E1 -396.094,E2 -396.094} C_VEL
LIN {X 0,Y 608.425,Z 676.693,A -85,B 0,C 180,E1 -398.591,E2 -398.591} C_VEL
LIN {X 0,Y 608.388,Z 676.694,A -85,B 0,C 180,E1 -401.182,E2 -401.182} C_VEL
LIN {X 0,Y 608.409,Z 676.692,A -85,B 0,C 180,E1 -403.313,E2 -403.313} C_VEL
LIN {X 0,Y 608.434,Z 676.696,A -85,B 0,C 180,E1 -406.137,E2 -406.137} C_VEL
LIN {X 0,Y 608.435,Z 676.693,A -85,B 0,C 180,E1 -408.831,E2 -408.831} C_VEL
LIN {X 0,Y 608.393,Z 676.694,A -85,B 0,C 180,E1 -411.415,E2 -411.415} C_VEL
LIN {X 0,Y 608.424,Z 676.693,A -85,B 0,C 180,E1 -413.091,E2 -413.091} C_VEL
LIN {X 0,Y 608.42,Z 676.69,A -85,B 0,C 180,E1 -415.536,E2 -415.536} C_VEL
LIN {X 0,Y 608.413,Z 676.692,A -85,B 0,C 180,E1 -417.91,E2 -417.91} C_VEL
LIN {X 0,Y 608.418,Z 676.693,A -85,B 0,C 180,E1 -420.225,E2 -420.225} C_VEL
LIN {X 0,Y 608.475,Z 676.695,A -85,B 0,C 180,E1 -422.794,E2 -422.794} C_VEL
LIN {X 0,Y 608.426,Z 676.779,A -85,B 0,C 180,E1 -423.855,E2 -423.855} C_VEL
LIN {X 0,Y 608.676,Z 680.188,A -85,B 0,C 180,E1 -424.24,E2 -424.24} C_VEL
LIN {X 0,Y 608.659,Z 706.573,A -85,B 0,C 180,E1 -427.089,E2 -427.089} C_VEL
LIN {X 0,Y 608.597,Z 731.618,A -85,B 0,C 180,E1 -429.737,E2 -429.737} C_VEL
LIN {X 0,Y 608.55,Z 756.832,A -85,B 0,C 180,E1 -432.359,E2 -432.359} C_VEL
LIN {X 0,Y 608.494,Z 782.045,A -85,B 0,C 180,E1 -434.943,E2 -434.943} C_VEL
LIN {X 0,Y 608.448,Z 801.916,A -85,B 0,C 180,E1 -436.957,E2 -436.957} C_VEL
LIN {X 0,Y 608.498,Z 912.233,A -85,B 0,C 180,E1 -438.281,E2 -438.281} C_VEL
LIN {X 0,Y 608.476,Z 925.405,A -85,B 0,C 180,E1 -438.576,E2 -438.576} C_VEL
LIN {X 0,Y 608.505,Z 937.727,A -85,B 0,C 180,E1 -438.986,E2 -438.986} C_VEL
LIN {X 0,Y 608.513,Z 949.734,A -85,B 0,C 180,E1 -439.525,E2 -439.525} C_VEL
LIN {X 0,Y 608.471,Z 961.275,A -85,B 0,C 180,E1 -440.196,E2 -440.196} C_VEL
LIN {X 0,Y 608.484,Z 971.658,A -85,B 0,C 180,E1 -440.951,E2 -440.951} C_VEL
LIN {X 0,Y 608.474,Z 980.051,A -85,B 0,C 180,E1 -441.704,E2 -441.704} C_VEL
LIN {X 0,Y 608.469,Z 988.003,A -85,B 0,C 180,E1 -442.539,E2 -442.539} C_VEL
LIN {X 0,Y 608.433,Z 995.318,A -85,B 0,C 180,E1 -443.489,E2 -443.489} C_VEL
LIN {X 0,Y 608.45,Z 1000.892,A -85,B 0,C 180,E1 -444.37,E2 -444.37} C_VEL
LIN {X 0,Y 608.432,Z 1005.97,A -85,B 0,C 180,E1 -445.367,E2 -445.367} C_VEL
LIN {X 0,Y 608.449,Z 1009.912,A -85,B 0,C 180,E1 -446.362,E2 -446.362} C_VEL
LIN {X 0,Y 608.425,Z 1012.821,A -85,B 0,C 180,E1 -447.356,E2 -447.356} C_VEL
LIN {X 0,Y 608.442,Z 1014.209,A -85,B 0,C 180,E1 -448.019,E2 -448.019} C_VEL
LIN {X 0,Y 608.438,Z 1015.787,A -85,B 0,C 180,E1 -449.343,E2 -449.343} C_VEL
LIN {X 0,Y 608.434,Z 1016,A -85,B 0,C 180,E1 -450.004,E2 -450.004} C_VEL
LIN {X 0,Y 608.448,Z 1015.179,A -85,B 0,C 180,E1 -451.328,E2 -451.328} C_VEL
LIN {X 0,Y 608.442,Z 1014.194,A -85,B 0,C 180,E1 -451.99,E2 -451.99} C_VEL
LIN {X 0,Y 608.425,Z 1012.798,A -85,B 0,C 180,E1 -452.652,E2 -452.652} C_VEL
LIN {X 0,Y 608.449,Z 1009.882,A -85,B 0,C 180,E1 -453.647,E2 -453.647} C_VEL
LIN {X 0,Y 608.432,Z 1005.932,A -85,B 0,C 180,E1 -454.642,E2 -454.642} C_VEL
LIN {X 0,Y 608.437,Z 999.852,A -85,B 0,C 180,E1 -455.805,E2 -455.805} C_VEL
LIN {X 0,Y 608.464,Z 993.206,A -85,B 0,C 180,E1 -456.803,E2 -456.803} C_VEL
LIN {X 0,Y 608.456,Z 984.954,A -85,B 0,C 180,E1 -457.804,E2 -457.804} C_VEL
LIN {X 0,Y 608.477,Z 974.554,A -85,B 0,C 180,E1 -458.807,E2 -458.807} C_VEL
LIN {X 0,Y 608.488,Z 963.691,A -85,B 0,C 180,E1 -459.645,E2 -459.645} C_VEL
LIN {X 0,Y 608.492,Z 952.703,A -85,B 0,C 180,E1 -460.317,E2 -460.317} C_VEL
LIN {X 0,Y 608.526,Z 940.912,A -85,B 0,C 180,E1 -460.884,E2 -460.884} C_VEL
LIN {X 0,Y 608.498,Z 928.767,A -85,B 0,C 180,E1 -461.327,E2 -461.327} C_VEL
LIN {X 0,Y 608.49,Z 916.315,A -85,B 0,C 180,E1 -461.644,E2 -461.644} C_VEL
LIN {X 0,Y 608.507,Z 900.423,A -85,B 0,C 180,E1 -461.876,E2 -461.876} C_VEL
LIN {X 0,Y 608.461,Z 802.051,A -85,B 0,C 180,E1 -463.041,E2 -463.041} C_VEL
LIN {X 0,Y 608.473,Z 778.594,A -85,B 0,C 180,E1 -465.409,E2 -465.409} C_VEL
LIN {X 0,Y 608.559,Z 753.381,A -85,B 0,C 180,E1 -467.998,E2 -467.998} C_VEL
LIN {X 0,Y 608.612,Z 726.679,A -85,B 0,C 180,E1 -470.782,E2 -470.782} C_VEL
LIN {X 0,Y 608.67,Z 699.592,A -85,B 0,C 180,E1 -473.659,E2 -473.659} C_VEL
LIN {X 0,Y 608.681,Z 679.592,A -85,B 0,C 180,E1 -475.825,E2 -475.825} C_VEL
LIN {X 0,Y 608.414,Z 676.694,A -85,B 0,C 180,E1 -476.178,E2 -476.178} C_VEL
LIN {X 0,Y 608.44,Z 676.692,A -85,B 0,C 180,E1 -478.614,E2 -478.614} C_VEL
LIN {X 0,Y 608.442,Z 676.696,A -85,B 0,C 180,E1 -481.321,E2 -481.321} C_VEL
LIN {X 0,Y 608.411,Z 676.694,A -85,B 0,C 180,E1 -483.726,E2 -483.726} C_VEL
LIN {X 0,Y 608.39,Z 676.695,A -85,B 0,C 180,E1 -486.099,E2 -486.099} C_VEL
LIN {X 0,Y 608.385,Z 676.695,A -85,B 0,C 180,E1 -488.23,E2 -488.23} C_VEL
LIN {X 0,Y 608.415,Z 676.692,A -85,B 0,C 180,E1 -490.325,E2 -490.325} C_VEL
LIN {X 0,Y 608.432,Z 676.696,A -85,B 0,C 180,E1 -492.964,E2 -492.964} C_VEL
LIN {X 0,Y 608.434,Z 676.692,A -85,B 0,C 180,E1 -495.741,E2 -495.741} C_VEL
LIN {X 0,Y 608.442,Z 676.689,A -85,B 0,C 180,E1 -497.937,E2 -497.937} C_VEL
LIN {X 0,Y 608.425,Z 676.693,A -85,B 0,C 180,E1 -500.71,E2 -500.71} C_VEL
LIN {X 0,Y 608.44,Z 676.696,A -85,B 0,C 180,E1 -503.084,E2 -503.084} C_VEL
LIN {X 0,Y 608.474,Z 676.691,A -85,B 0,C 180,E1 -505.531,E2 -505.531} C_VEL
LIN {X 0,Y 608.464,Z 676.687,A -85,B 0,C 180,E1 -507.905,E2 -507.905} C_VEL
LIN {X 0,Y 608.464,Z 676.685,A -85,B 0,C 180,E1 -510.22,E2 -510.22} C_VEL
LIN {X 0,Y 608.443,Z 676.691,A -85,B 0,C 180,E1 -512.801,E2 -512.801} C_VEL
LIN {X 0,Y 608.448,Z 676.697,A -85,B 0,C 180,E1 -515.429,E2 -515.429} C_VEL
LIN {X 0,Y 608.463,Z 676.686,A -85,B 0,C 180,E1 -518.308,E2 -518.308} C_VEL
LIN {X 0,Y 608.477,Z 676.693,A -85,B 0,C 180,E1 -521.284,E2 -521.284} C_VEL
LIN {X 0,Y 608.454,Z 676.69,A -85,B 0,C 180,E1 -523.906,E2 -523.906} C_VEL
LIN {X 0,Y 608.46,Z 676.687,A -85,B 0,C 180,E1 -526.643,E2 -526.643} C_VEL
LIN {X 0,Y 608.466,Z 676.694,A -85,B 0,C 180,E1 -527.291,E2 -527.291} C_VEL
LIN {X 0,Y 608.539,Z 761.772,A -85,B 0,C 180,E1 -528.319,E2 -528.319} C_VEL
LIN {X 0,Y 608.538,Z 775.113,A -85,B 0,C 180,E1 -528.614,E2 -528.614} C_VEL
LIN {X 0,Y 608.521,Z 788.484,A -85,B 0,C 180,E1 -529.059,E2 -529.059} C_VEL
LIN {X 0,Y 608.495,Z 800.36,A -85,B 0,C 180,E1 -529.603,E2 -529.603} C_VEL
LIN {X 0,Y 608.486,Z 811.782,A -85,B 0,C 180,E1 -530.275,E2 -530.275} C_VEL
LIN {X 0,Y 608.474,Z 822.08,A -85,B 0,C 180,E1 -531.029,E2 -531.029} C_VEL
LIN {X 0,Y 608.464,Z 831.243,A -85,B 0,C 180,E1 -531.866,E2 -531.866} C_VEL
LIN {X 0,Y 608.462,Z 838.965,A -85,B 0,C 180,E1 -532.701,E2 -532.701} C_VEL
LIN {X 0,Y 608.448,Z 846.435,A -85,B 0,C 180,E1 -533.7,E2 -533.7} C_VEL
LIN {X 0,Y 608.462,Z 852.433,A -85,B 0,C 180,E1 -534.698,E2 -534.698} C_VEL
LIN {X 0,Y 608.439,Z 857.177,A -85,B 0,C 180,E1 -535.694,E2 -535.694} C_VEL
LIN {X 0,Y 608.426,Z 860.811,A -85,B 0,C 180,E1 -536.689,E2 -536.689} C_VEL
LIN {X 0,Y 608.425,Z 862.691,A -85,B 0,C 180,E1 -537.352,E2 -537.352} C_VEL
LIN {X 0,Y 608.442,Z 864.127,A -85,B 0,C 180,E1 -538.014,E2 -538.014} C_VEL
LIN {X 0,Y 608.439,Z 865.752,A -85,B 0,C 180,E1 -539.338,E2 -539.338} C_VEL
LIN {X 0,Y 608.435,Z 865.995,A -85,B 0,C 180,E1 -540,E2 -540} C_VEL
LIN {X 0,Y 608.438,Z 865.815,A -85,B 0,C 180,E1 -540.662,E2 -540.662} C_VEL
LIN {X 0,Y 608.441,Z 864.276,A -85,B 0,C 180,E1 -541.986,E2 -541.986} C_VEL
LIN {X 0,Y 608.426,Z 862.917,A -85,B 0,C 180,E1 -542.648,E2 -542.648} C_VEL
LIN {X 0,Y 608.449,Z 860.04,A -85,B 0,C 180,E1 -543.642,E2 -543.642} C_VEL
LIN {X 0,Y 608.433,Z 856.141,A -85,B 0,C 180,E1 -544.638,E2 -544.638} C_VEL
LIN {X 0,Y 608.449,Z 851.111,A -85,B 0,C 180,E1 -545.634,E2 -545.634} C_VEL
LIN {X 0,Y 608.441,Z 844.794,A -85,B 0,C 180,E1 -546.633,E2 -546.633} C_VEL
LIN {X 0,Y 608.476,Z 836.877,A -85,B 0,C 180,E1 -547.633,E2 -547.633} C_VEL
LIN {X 0,Y 608.472,Z 827.029,A -85,B 0,C 180,E1 -548.636,E2 -548.636} C_VEL
LIN {X 0,Y 608.477,Z 824.972,A -85,B 0,C 180,E1 -548.816,E2 -548.816} C_VEL
LIN {X 0,Y 607.804,Z 820.637,A -85,B 0,C 180,E1 -549.187,E2 -549.187} C_VEL
LIN {X 0,Y 604.941,Z 813.394,A -85,B 0,C 180,E1 -549.766,E2 -549.766} C_VEL
LIN {X 0,Y 602.122,Z 805.767,A -85,B 0,C 180,E1 -550.298,E2 -550.298} C_VEL
LIN {X 0,Y 601.519,Z 800.688,A -85,B 0,C 180,E1 -550.591,E2 -550.591} C_VEL
LIN {X 0,Y 601.546,Z 788.829,A -85,B 0,C 180,E1 -551.146,E2 -551.146} C_VEL
LIN {X 0,Y 601.594,Z 776.057,A -85,B 0,C 180,E1 -551.583,E2 -551.583} C_VEL
LIN {X 0,Y 601.605,Z 763.197,A -85,B 0,C 180,E1 -551.882,E2 -551.882} C_VEL
LIN {X 0,Y 601.589,Z 725.864,A -85,B 0,C 180,E1 -552.353,E2 -552.353} C_VEL
LIN {X 0,Y 601.536,Z 678.231,A -85,B 0,C 180,E1 -552.925,E2 -552.925} C_VEL
LIN {X 0,Y 601.434,Z 677.568,A -85,B 0,C 180,E1 -552.957,E2 -552.957} C_VEL
LIN {X 0,Y 601.409,Z 677.565,A -85,B 0,C 180,E1 -555.592,E2 -555.592} C_VEL
LIN {X 0,Y 601.391,Z 677.567,A -85,B 0,C 180,E1 -557.689,E2 -557.689} C_VEL
LIN {X 0,Y 601.427,Z 677.569,A -85,B 0,C 180,E1 -560.522,E2 -560.522} C_VEL
LIN {X 0,Y 601.4,Z 677.567,A -85,B 0,C 180,E1 -563.411,E2 -563.411} C_VEL
LIN {X 0,Y 601.412,Z 677.564,A -85,B 0,C 180,E1 -565.865,E2 -565.865} C_VEL
LIN {X 0,Y 601.431,Z 677.568,A -85,B 0,C 180,E1 -568.627,E2 -568.627} C_VEL
LIN {X 0,Y 601.424,Z 677.565,A -85,B 0,C 180,E1 -571.453,E2 -571.453} C_VEL
LIN {X 0,Y 601.428,Z 677.562,A -85,B 0,C 180,E1 -574.119,E2 -574.119} C_VEL
LIN {X 0,Y 601.441,Z 677.564,A -85,B 0,C 180,E1 -577.381,E2 -577.381} C_VEL
LIN {X 0,Y 601.408,Z 677.564,A -85,B 0,C 180,E1 -579.996,E2 -579.996} C_VEL
LIN {X 0,Y 601.419,Z 677.568,A -85,B 0,C 180,E1 -582.67,E2 -582.67} C_VEL
LIN {X 0,Y 601.412,Z 677.567,A -85,B 0,C 180,E1 -585.478,E2 -585.478} C_VEL
LIN {X 0,Y 601.423,Z 677.564,A -85,B 0,C 180,E1 -588.407,E2 -588.407} C_VEL
LIN {X 0,Y 601.406,Z 677.571,A -85,B 0,C 180,E1 -590.871,E2 -590.871} C_VEL
LIN {X 0,Y 601.397,Z 677.572,A -85,B 0,C 180,E1 -593.414,E2 -593.414} C_VEL
LIN {X 0,Y 601.382,Z 677.568,A -85,B 0,C 180,E1 -596.072,E2 -596.072} C_VEL
LIN {X 0,Y 601.398,Z 677.567,A -85,B 0,C 180,E1 -598.549,E2 -598.549} C_VEL
LIN {X 0,Y 601.418,Z 677.572,A -85,B 0,C 180,E1 -601.37,E2 -601.37} C_VEL
LIN {X 0,Y 601.353,Z 677.571,A -85,B 0,C 180,E1 -604.145,E2 -604.145} C_VEL
LIN {X 0,Y 601.357,Z 677.572,A -85,B 0,C 180,E1 -606.584,E2 -606.584} C_VEL
LIN {X 0,Y 601.413,Z 677.572,A -85,B 0,C 180,E1 -609.474,E2 -609.474} C_VEL
LIN {X 0,Y 601.376,Z 677.575,A -85,B 0,C 180,E1 -611.603,E2 -611.603} C_VEL
LIN {X 0,Y 601.417,Z 677.569,A -85,B 0,C 180,E1 -613.709,E2 -613.709} C_VEL
LIN {X 0,Y 601.365,Z 677.57,A -85,B 0,C 180,E1 -616.479,E2 -616.479} C_VEL
LIN {X 0,Y 601.41,Z 677.571,A -85,B 0,C 180,E1 -617.147,E2 -617.147} C_VEL
LIN {X 0,Y 601.656,Z 682.281,A -85,B 0,C 180,E1 -617.216,E2 -617.216} C_VEL
LIN {X 0,Y 601.539,Z 762.773,A -85,B 0,C 180,E1 -618.198,E2 -618.198} C_VEL
LIN {X 0,Y 601.524,Z 776.533,A -85,B 0,C 180,E1 -618.519,E2 -618.519} C_VEL
LIN {X 0,Y 601.507,Z 788.977,A -85,B 0,C 180,E1 -618.95,E2 -618.95} C_VEL
LIN {X 0,Y 601.526,Z 800.287,A -85,B 0,C 180,E1 -619.478,E2 -619.478} C_VEL
LIN {X 0,Y 601.46,Z 811.717,A -85,B 0,C 180,E1 -620.157,E2 -620.157} C_VEL
LIN {X 0,Y 601.439,Z 822.019,A -85,B 0,C 180,E1 -620.92,E2 -620.92} C_VEL
LIN {X 0,Y 601.404,Z 831.221,A -85,B 0,C 180,E1 -621.766,E2 -621.766} C_VEL
LIN {X 0,Y 601.414,Z 838.943,A -85,B 0,C 180,E1 -622.611,E2 -622.611} C_VEL
LIN {X 0,Y 601.361,Z 846.334,A -85,B 0,C 180,E1 -623.609,E2 -623.609} C_VEL
LIN {X 0,Y 601.373,Z 852.42,A -85,B 0,C 180,E1 -624.631,E2 -624.631} C_VEL
LIN {X 0,Y 601.354,Z 857.166,A -85,B 0,C 180,E1 -625.639,E2 -625.639} C_VEL
LIN {X 0,Y 601.344,Z 860.803,A -85,B 0,C 180,E1 -626.646,E2 -626.646} C_VEL
LIN {X 0,Y 601.324,Z 862.679,A -85,B 0,C 180,E1 -627.316,E2 -627.316} C_VEL
LIN {X 0,Y 601.341,Z 864.113,A -85,B 0,C 180,E1 -627.986,E2 -627.986} C_VEL
LIN {X 0,Y 601.347,Z 865.127,A -85,B 0,C 180,E1 -628.656,E2 -628.656} C_VEL
LIN {X 0,Y 601.336,Z 865.986,A -85,B 0,C 180,E1 -629.996,E2 -629.996} C_VEL
LIN {X 0,Y 601.339,Z 865.818,A -85,B 0,C 180,E1 -630.665,E2 -630.665} C_VEL
LIN {X 0,Y 601.341,Z 864.282,A -85,B 0,C 180,E1 -632.005,E2 -632.005} C_VEL
LIN {X 0,Y 601.326,Z 862.928,A -85,B 0,C 180,E1 -632.675,E2 -632.675} C_VEL
LIN {X 0,Y 601.367,Z 860.057,A -85,B 0,C 180,E1 -633.681,E2 -633.681} C_VEL
LIN {X 0,Y 601.337,Z 856.164,A -85,B 0,C 180,E1 -634.688,E2 -634.688} C_VEL
LIN {X 0,Y 601.372,Z 851.14,A -85,B 0,C 180,E1 -635.696,E2 -635.696} C_VEL
LIN {X 0,Y 601.376,Z 844.821,A -85,B 0,C 180,E1 -636.706,E2 -636.706} C_VEL
LIN {X 0,Y 601.394,Z 836.901,A -85,B 0,C 180,E1 -637.718,E2 -637.718} C_VEL
LIN {X 0,Y 601.421,Z 828.818,A -85,B 0,C 180,E1 -638.563,E2 -638.563} C_VEL
LIN {X 0,Y 601.451,Z 819.019,A -85,B 0,C 180,E1 -639.41,E2 -639.41} C_VEL
LIN {X 0,Y 601.486,Z 808.011,A -85,B 0,C 180,E1 -640.174,E2 -640.174} C_VEL
LIN {X 0,Y 601.528,Z 795.677,A -85,B 0,C 180,E1 -640.844,E2 -640.844} C_VEL
LIN {X 0,Y 601.498,Z 783.842,A -85,B 0,C 180,E1 -641.335,E2 -641.335} C_VEL
LIN {X 0,Y 601.518,Z 771.47,A -85,B 0,C 180,E1 -641.707,E2 -641.707} C_VEL
LIN {X 0,Y 601.549,Z 758.138,A -85,B 0,C 180,E1 -641.963,E2 -641.963} C_VEL
LIN {X 0,Y 601.581,Z 678.471,A -85,B 0,C 180,E1 -642.921,E2 -642.921} C_VEL
LIN {X 0,Y 601.412,Z 677.571,A -85,B 0,C 180,E1 -642.952,E2 -642.952} C_VEL
LIN {X 0,Y 601.373,Z 677.569,A -85,B 0,C 180,E1 -645.587,E2 -645.587} C_VEL
LIN {X 0,Y 601.358,Z 677.571,A -85,B 0,C 180,E1 -647.684,E2 -647.684} C_VEL
LIN {X 0,Y 601.367,Z 677.569,A -85,B 0,C 180,E1 -649.805,E2 -649.805} C_VEL
LIN {X 0,Y 601.366,Z 677.569,A -85,B 0,C 180,E1 -651.955,E2 -651.955} C_VEL
LIN {X 0,Y 601.38,Z 677.575,A -85,B 0,C 180,E1 -654.873,E2 -654.873} C_VEL
LIN {X 0,Y 601.399,Z 677.572,A -85,B 0,C 180,E1 -657.359,E2 -657.359} C_VEL
LIN {X 0,Y 601.368,Z 677.569,A -85,B 0,C 180,E1 -660.138,E2 -660.138} C_VEL
LIN {X 0,Y 601.381,Z 677.569,A -85,B 0,C 180,E1 -662.709,E2 -662.709} C_VEL
LIN {X 0,Y 601.38,Z 677.574,A -85,B 0,C 180,E1 -665.109,E2 -665.109} C_VEL
LIN {X 0,Y 601.401,Z 677.576,A -85,B 0,C 180,E1 -667.413,E2 -667.413} C_VEL
LIN {X 0,Y 601.37,Z 677.572,A -85,B 0,C 180,E1 -669.989,E2 -669.989} C_VEL
LIN {X 0,Y 601.359,Z 677.57,A -85,B 0,C 180,E1 -672.585,E2 -672.585} C_VEL
LIN {X 0,Y 601.374,Z 677.568,A -85,B 0,C 180,E1 -674.53,E2 -674.53} C_VEL
LIN {X 0,Y 601.41,Z 677.569,A -85,B 0,C 180,E1 -677.399,E2 -677.399} C_VEL
LIN {X 0,Y 601.387,Z 677.568,A -85,B 0,C 180,E1 -680.459,E2 -680.459} C_VEL
LIN {X 0,Y 601.376,Z 677.569,A -85,B 0,C 180,E1 -682.613,E2 -682.613} C_VEL
LIN {X 0,Y 601.371,Z 677.568,A -85,B 0,C 180,E1 -685.065,E2 -685.065} C_VEL
LIN {X 0,Y 601.382,Z 677.569,A -85,B 0,C 180,E1 -687.481,E2 -687.481} C_VEL
LIN {X 0,Y 601.429,Z 677.568,A -85,B 0,C 180,E1 -689.836,E2 -689.836} C_VEL
LIN {X 0,Y 601.384,Z 677.568,A -85,B 0,C 180,E1 -692.885,E2 -692.885} C_VEL
LIN {X 0,Y 601.346,Z 677.572,A -85,B 0,C 180,E1 -695.119,E2 -695.119} C_VEL
LIN {X 0,Y 601.341,Z 677.572,A -85,B 0,C 180,E1 -697.391,E2 -697.391} C_VEL
LIN {X 0,Y 601.36,Z 677.57,A -85,B 0,C 180,E1 -699.476,E2 -699.476} C_VEL
LIN {X 0,Y 601.369,Z 677.577,A -85,B 0,C 180,E1 -702.311,E2 -702.311} C_VEL
LIN {X 0,Y 601.368,Z 677.571,A -85,B 0,C 180,E1 -705.101,E2 -705.101} C_VEL
LIN {X 0,Y 601.352,Z 677.571,A -85,B 0,C 180,E1 -707.856,E2 -707.856} C_VEL
LIN {X 0,Y 601.392,Z 677.575,A -85,B 0,C 180,E1 -710.584,E2 -710.584} C_VEL
LIN {X 0,Y 601.371,Z 677.571,A -85,B 0,C 180,E1 -713.322,E2 -713.322} C_VEL
LIN {X 0,Y 601.366,Z 677.572,A -85,B 0,C 180,E1 -715.308,E2 -715.308} C_VEL
LIN {X 0,Y 601.385,Z 677.571,A -85,B 0,C 180,E1 -717.321,E2 -717.321} C_VEL
LIN {X 0,Y 601.36,Z 677.57,A -85,B 0,C 180,E1 -720,E2 -720} C_VEL
LIN {X 0,Y 601.386,Z 677.571,A -85,B 0,C 180,E1 -722.679,E2 -722.679} C_VEL
LIN {X 0,Y 601.418,Z 677.57,A -85,B 0,C 180,E1 -725.364,E2 -725.364} C_VEL
LIN {X 0,Y 601.368,Z 677.569,A -85,B 0,C 180,E1 -728.062,E2 -728.062} C_VEL
LIN {X 0,Y 601.362,Z 677.572,A -85,B 0,C 180,E1 -730.777,E2 -730.777} C_VEL
LIN {X 0,Y 601.374,Z 677.577,A -85,B 0,C 180,E1 -733.517,E2 -733.517} C_VEL
LIN {X 0,Y 601.381,Z 677.568,A -85,B 0,C 180,E1 -736.289,E2 -736.289} C_VEL
LIN {X 0,Y 601.361,Z 677.573,A -85,B 0,C 180,E1 -739.101,E2 -739.101} C_VEL
LIN {X 0,Y 601.366,Z 677.575,A -85,B 0,C 180,E1 -741.961,E2 -741.961} C_VEL
LIN {X 0,Y 601.388,Z 677.568,A -85,B 0,C 180,E1 -744.302,E2 -744.302} C_VEL
LIN {X 0,Y 601.356,Z 677.572,A -85,B 0,C 180,E1 -746.366,E2 -746.366} C_VEL
LIN {X 0,Y 601.375,Z 677.568,A -85,B 0,C 180,E1 -748.794,E2 -748.794} C_VEL
LIN {X 0,Y 601.372,Z 677.568,A -85,B 0,C 180,E1 -750.945,E2 -750.945} C_VEL
LIN {X 0,Y 601.38,Z 677.569,A -85,B 0,C 180,E1 -753.317,E2 -753.317} C_VEL
LIN {X 0,Y 601.391,Z 677.574,A -85,B 0,C 180,E1 -756.272,E2 -756.272} C_VEL
LIN {X 0,Y 601.378,Z 677.567,A -85,B 0,C 180,E1 -759.129,E2 -759.129} C_VEL
LIN {X 0,Y 601.385,Z 677.57,A -85,B 0,C 180,E1 -761.769,E2 -761.769} C_VEL
LIN {X 0,Y 601.373,Z 677.576,A -85,B 0,C 180,E1 -764.54,E2 -764.54} C_VEL
LIN {X 0,Y 601.36,Z 677.57,A -85,B 0,C 180,E1 -767.335,E2 -767.335} C_VEL
LIN {X 0,Y 601.367,Z 677.569,A -85,B 0,C 180,E1 -769.432,E2 -769.432} C_VEL
LIN {X 0,Y 601.366,Z 677.57,A -85,B 0,C 180,E1 -771.737,E2 -771.737} C_VEL
LIN {X 0,Y 601.351,Z 677.576,A -85,B 0,C 180,E1 -774.251,E2 -774.251} C_VEL
LIN {X 0,Y 601.398,Z 677.576,A -85,B 0,C 180,E1 -776.693,E2 -776.693} C_VEL
LIN {X 0,Y 601.394,Z 677.572,A -85,B 0,C 180,E1 -779.064,E2 -779.064} C_VEL
LIN {X 0,Y 601.397,Z 677.569,A -85,B 0,C 180,E1 -781.379,E2 -781.379} C_VEL
LIN {X 0,Y 601.389,Z 677.62,A -85,B 0,C 180,E1 -783.619,E2 -783.619} C_VEL
LIN {X 0,Y 601.912,Z 681.151,A -85,B 0,C 180,E1 -784.035,E2 -784.035} C_VEL
LIN {X 0,Y 601.845,Z 706.573,A -85,B 0,C 180,E1 -786.814,E2 -786.814} C_VEL
LIN {X 0,Y 601.741,Z 731.618,A -85,B 0,C 180,E1 -789.495,E2 -789.495} C_VEL
LIN {X 0,Y 601.615,Z 758.513,A -85,B 0,C 180,E1 -792.324,E2 -792.324} C_VEL
LIN {X 0,Y 601.509,Z 785.407,A -85,B 0,C 180,E1 -795.111,E2 -795.111} C_VEL
LIN {X 0,Y 601.445,Z 801.916,A -85,B 0,C 180,E1 -796.802,E2 -796.802} C_VEL
LIN {X 0,Y 601.611,Z 877.931,A -85,B 0,C 180,E1 -797.717,E2 -797.717} C_VEL
LIN {X 0,Y 601.57,Z 912.233,A -85,B 0,C 180,E1 -798.144,E2 -798.144} C_VEL
LIN {X 0,Y 601.539,Z 925.405,A -85,B 0,C 180,E1 -798.442,E2 -798.442} C_VEL
LIN {X 0,Y 601.533,Z 937.012,A -85,B 0,C 180,E1 -798.829,E2 -798.829} C_VEL
LIN {X 0,Y 601.52,Z 949.733,A -85,B 0,C 180,E1 -799.401,E2 -799.401} C_VEL
LIN {X 0,Y 601.471,Z 961.276,A -85,B 0,C 180,E1 -800.081,E2 -800.081} C_VEL
LIN {X 0,Y 601.458,Z 971.659,A -85,B 0,C 180,E1 -800.844,E2 -800.844} C_VEL
LIN {X 0,Y 601.428,Z 980.06,A -85,B 0,C 180,E1 -801.606,E2 -801.606} C_VEL
LIN {X 0,Y 601.415,Z 988.003,A -85,B 0,C 180,E1 -802.451,E2 -802.451} C_VEL
LIN {X 0,Y 601.361,Z 995.274,A -85,B 0,C 180,E1 -803.405,E2 -803.405} C_VEL
LIN {X 0,Y 601.373,Z 1000.893,A -85,B 0,C 180,E1 -804.304,E2 -804.304} C_VEL
LIN {X 0,Y 601.336,Z 1005.97,A -85,B 0,C 180,E1 -805.312,E2 -805.312} C_VEL
LIN {X 0,Y 601.367,Z 1009.911,A -85,B 0,C 180,E1 -806.319,E2 -806.319} C_VEL
LIN {X 0,Y 601.325,Z 1012.821,A -85,B 0,C 180,E1 -807.325,E2 -807.325} C_VEL
LIN {X 0,Y 601.341,Z 1014.209,A -85,B 0,C 180,E1 -807.995,E2 -807.995} C_VEL
LIN {X 0,Y 601.339,Z 1015.787,A -85,B 0,C 180,E1 -809.335,E2 -809.335} C_VEL
LIN {X 0,Y 601.335,Z 1016,A -85,B 0,C 180,E1 -810.004,E2 -810.004} C_VEL
LIN {X 0,Y 601.347,Z 1015.179,A -85,B 0,C 180,E1 -811.344,E2 -811.344} C_VEL
LIN {X 0,Y 601.341,Z 1014.194,A -85,B 0,C 180,E1 -812.014,E2 -812.014} C_VEL
LIN {X 0,Y 601.325,Z 1012.798,A -85,B 0,C 180,E1 -812.684,E2 -812.684} C_VEL
LIN {X 0,Y 601.368,Z 1009.882,A -85,B 0,C 180,E1 -813.69,E2 -813.69} C_VEL
LIN {X 0,Y 601.336,Z 1005.932,A -85,B 0,C 180,E1 -814.697,E2 -814.697} C_VEL
LIN {X 0,Y 601.372,Z 999.852,A -85,B 0,C 180,E1 -815.873,E2 -815.873} C_VEL
LIN {X 0,Y 601.385,Z 993.206,A -85,B 0,C 180,E1 -816.884,E2 -816.884} C_VEL
LIN {X 0,Y 601.402,Z 984.955,A -85,B 0,C 180,E1 -817.896,E2 -817.896} C_VEL
LIN {X 0,Y 601.436,Z 974.554,A -85,B 0,C 180,E1 -818.911,E2 -818.911} C_VEL
LIN {X 0,Y 601.461,Z 963.691,A -85,B 0,C 180,E1 -819.759,E2 -819.759} C_VEL
LIN {X 0,Y 601.495,Z 952.704,A -85,B 0,C 180,E1 -820.438,E2 -820.438} C_VEL
LIN {X 0,Y 601.539,Z 940.79,A -85,B 0,C 180,E1 -821.017,E2 -821.017} C_VEL
LIN {X 0,Y 601.522,Z 928.766,A -85,B 0,C 180,E1 -821.46,E2 -821.46} C_VEL
LIN {X 0,Y 601.561,Z 916.315,A -85,B 0,C 180,E1 -821.78,E2 -821.78} C_VEL
LIN {X 0,Y 601.587,Z 900.423,A -85,B 0,C 180,E1 -822.014,E2 -822.014} C_VEL
LIN {X 0,Y 601.471,Z 802.051,A -85,B 0,C 180,E1 -823.196,E2 -823.196} C_VEL
LIN {X 0,Y 601.504,Z 778.594,A -85,B 0,C 180,E1 -825.592,E2 -825.592} C_VEL
LIN {X 0,Y 601.652,Z 753.381,A -85,B 0,C 180,E1 -828.212,E2 -828.212} C_VEL
LIN {X 0,Y 601.772,Z 724.806,A -85,B 0,C 180,E1 -831.229,E2 -831.229} C_VEL
LIN {X 0,Y 601.866,Z 699.592,A -85,B 0,C 180,E1 -833.943,E2 -833.943} C_VEL
LIN {X 0,Y 601.893,Z 680.07,A -85,B 0,C 180,E1 -836.085,E2 -836.085} C_VEL
LIN {X 0,Y 601.37,Z 677.576,A -85,B 0,C 180,E1 -836.415,E2 -836.415} C_VEL
LIN {X 0,Y 601.404,Z 677.571,A -85,B 0,C 180,E1 -838.783,E2 -838.783} C_VEL
LIN {X 0,Y 601.376,Z 677.57,A -85,B 0,C 180,E1 -841.731,E2 -841.731} C_VEL
LIN {X 0,Y 601.343,Z 677.573,A -85,B 0,C 180,E1 -844.127,E2 -844.127} C_VEL
LIN {X 0,Y 601.374,Z 677.57,A -85,B 0,C 180,E1 -846.588,E2 -846.588} C_VEL
LIN {X 0,Y 601.398,Z 677.571,A -85,B 0,C 180,E1 -849.531,E2 -849.531} C_VEL
LIN {X 0,Y 601.402,Z 677.567,A -85,B 0,C 180,E1 -851.769,E2 -851.769} C_VEL
LIN {X 0,Y 601.377,Z 677.57,A -85,B 0,C 180,E1 -854.53,E2 -854.53} C_VEL
LIN {X 0,Y 601.396,Z 677.574,A -85,B 0,C 180,E1 -857.413,E2 -857.413} C_VEL
LIN {X 0,Y 601.404,Z 677.566,A -85,B 0,C 180,E1 -860.004,E2 -860.004} C_VEL
LIN {X 0,Y 601.397,Z 677.567,A -85,B 0,C 180,E1 -862.625,E2 -862.625} C_VEL
LIN {X 0,Y 601.409,Z 677.572,A -85,B 0,C 180,E1 -865.068,E2 -865.068} C_VEL
LIN {X 0,Y 601.435,Z 677.569,A -85,B 0,C 180,E1 -867.484,E2 -867.484} C_VEL
LIN {X 0,Y 601.416,Z 677.566,A -85,B 0,C 180,E1 -869.856,E2 -869.856} C_VEL
LIN {X 0,Y 601.403,Z 677.566,A -85,B 0,C 180,E1 -872.132,E2 -872.132} C_VEL
LIN {X 0,Y 601.413,Z 677.564,A -85,B 0,C 180,E1 -874.382,E2 -874.382} C_VEL
LIN {X 0,Y 601.397,Z 677.567,A -85,B 0,C 180,E1 -876.589,E2 -876.589} C_VEL
LIN {X 0,Y 601.432,Z 677.571,A -85,B 0,C 180,E1 -879.478,E2 -879.478} C_VEL
LIN {X 0,Y 601.392,Z 677.567,A -85,B 0,C 180,E1 -882.311,E2 -882.311} C_VEL
LIN {X 0,Y 601.41,Z 677.565,A -85,B 0,C 180,E1 -884.409,E2 -884.409} C_VEL
LIN {X 0,Y 601.423,Z 677.569,A -85,B 0,C 180,E1 -887.15,E2 -887.15} C_VEL
LIN {X 0,Y 601.659,Z 684.372,A -85,B 0,C 180,E1 -887.241,E2 -887.241} C_VEL
LIN {X 0,Y 601.613,Z 761.777,A -85,B 0,C 180,E1 -888.182,E2 -888.182} C_VEL
LIN {X 0,Y 601.581,Z 774.372,A -85,B 0,C 180,E1 -888.459,E2 -888.459} C_VEL
LIN {X 0,Y 601.537,Z 787.614,A -85,B 0,C 180,E1 -888.897,E2 -888.897} C_VEL
LIN {X 0,Y 601.534,Z 798.753,A -85,B 0,C 180,E1 -889.396,E2 -889.396} C_VEL
LIN {X 0,Y 601.442,Z 809.218,A -85,B 0,C 180,E1 -889.99,E2 -889.99} C_VEL
LIN {X 0,Y 601.432,Z 819.963,A -85,B 0,C 180,E1 -890.754,E2 -890.754} C_VEL
LIN {X 0,Y 601.425,Z 827.858,A -85,B 0,C 180,E1 -891.432,E2 -891.432} C_VEL
LIN {X 0,Y 601.418,Z 837.566,A -85,B 0,C 180,E1 -892.446,E2 -892.446} C_VEL
LIN {X 0,Y 601.373,Z 844.919,A -85,B 0,C 180,E1 -893.397,E2 -893.397} C_VEL
LIN {X 0,Y 601.372,Z 850.612,A -85,B 0,C 180,E1 -894.299,E2 -894.299} C_VEL
LIN {X 0,Y 601.335,Z 855.751,A -85,B 0,C 180,E1 -895.307,E2 -895.307} C_VEL
LIN {X 0,Y 601.367,Z 859.741,A -85,B 0,C 180,E1 -896.315,E2 -896.315} C_VEL
LIN {X 0,Y 601.324,Z 862.694,A -85,B 0,C 180,E1 -897.32,E2 -897.32} C_VEL
LIN {X 0,Y 601.341,Z 864.129,A -85,B 0,C 180,E1 -897.991,E2 -897.991} C_VEL
LIN {X 0,Y 601.339,Z 865.753,A -85,B 0,C 180,E1 -899.33,E2 -899.33} C_VEL
LIN {X 0,Y 601.335,Z 865.996,A -85,B 0,C 180,E1 -900,E2 -900} C_VEL
LIN {X 0,Y 601.339,Z 865.815,A -85,B 0,C 180,E1 -900.67,E2 -900.67} C_VEL
LIN {X 0,Y 601.34,Z 864.276,A -85,B 0,C 180,E1 -902.009,E2 -902.009} C_VEL
LIN {X 0,Y 601.326,Z 862.907,A -85,B 0,C 180,E1 -902.68,E2 -902.68} C_VEL
LIN {X 0,Y 601.368,Z 860.032,A -85,B 0,C 180,E1 -903.685,E2 -903.685} C_VEL
LIN {X 0,Y 601.337,Z 856.133,A -85,B 0,C 180,E1 -904.693,E2 -904.693} C_VEL
LIN {X 0,Y 601.373,Z 851.105,A -85,B 0,C 180,E1 -905.701,E2 -905.701} C_VEL
LIN {X 0,Y 601.362,Z 844.791,A -85,B 0,C 180,E1 -906.711,E2 -906.711} C_VEL
LIN {X 0,Y 601.397,Z 836.872,A -85,B 0,C 180,E1 -907.723,E2 -907.723} C_VEL
LIN {X 0,Y 601.417,Z 827.01,A -85,B 0,C 180,E1 -908.738,E2 -908.738} C_VEL
LIN {X 0,Y 601.443,Z 816.709,A -85,B 0,C 180,E1 -909.585,E2 -909.585} C_VEL
LIN {X 0,Y 601.48,Z 805.096,A -85,B 0,C 180,E1 -910.349,E2 -910.349} C_VEL
LIN {X 0,Y 601.519,Z 800.688,A -85,B 0,C 180,E1 -910.591,E2 -910.591} C_VEL
LIN {X 0,Y 600.937,Z 795.559,A -85,B 0,C 180,E1 -910.864,E2 -910.864} C_VEL
LIN {X 0,Y 598.2,Z 787.105,A -85,B 0,C 180,E1 -911.283,E2 -911.283} C_VEL
LIN {X 0,Y 595.369,Z 778.359,A -85,B 0,C 180,E1 -911.639,E2 -911.639} C_VEL
LIN {X 0,Y 594.639,Z 772.777,A -85,B 0,C 180,E1 -911.81,E2 -911.81} C_VEL
LIN {X 0,Y 594.662,Z 760.754,A -85,B 0,C 180,E1 -912.066,E2 -912.066} C_VEL
LIN {X 0,Y 594.657,Z 679.7,A -85,B 0,C 180,E1 -913.059,E2 -913.059} C_VEL
LIN {X 0,Y 594.392,Z 678.443,A -85,B 0,C 180,E1 -913.091,E2 -913.091} C_VEL
LIN {X 0,Y 594.362,Z 678.443,A -85,B 0,C 180,E1 -915.781,E2 -915.781} C_VEL
LIN {X 0,Y 594.379,Z 678.449,A -85,B 0,C 180,E1 -918.618,E2 -918.618} C_VEL
LIN {X 0,Y 594.363,Z 678.443,A -85,B 0,C 180,E1 -921.504,E2 -921.504} C_VEL
LIN {X 0,Y 594.398,Z 678.442,A -85,B 0,C 180,E1 -924.446,E2 -924.446} C_VEL
LIN {X 0,Y 594.368,Z 678.443,A -85,B 0,C 180,E1 -927.461,E2 -927.461} C_VEL
LIN {X 0,Y 594.395,Z 678.44,A -85,B 0,C 180,E1 -930.327,E2 -930.327} C_VEL
LIN {X 0,Y 594.385,Z 678.45,A -85,B 0,C 180,E1 -932.95,E2 -932.95} C_VEL
LIN {X 0,Y 594.338,Z 678.448,A -85,B 0,C 180,E1 -935.41,E2 -935.41} C_VEL
LIN {X 0,Y 594.388,Z 678.439,A -85,B 0,C 180,E1 -937.941,E2 -937.941} C_VEL
LIN {X 0,Y 594.377,Z 678.448,A -85,B 0,C 180,E1 -940.82,E2 -940.82} C_VEL
LIN {X 0,Y 594.362,Z 678.448,A -85,B 0,C 180,E1 -943.3,E2 -943.3} C_VEL
LIN {X 0,Y 594.356,Z 678.443,A -85,B 0,C 180,E1 -946.162,E2 -946.162} C_VEL
LIN {X 0,Y 594.373,Z 678.45,A -85,B 0,C 180,E1 -949.179,E2 -949.179} C_VEL
LIN {X 0,Y 594.323,Z 678.447,A -85,B 0,C 180,E1 -952.052,E2 -952.052} C_VEL
LIN {X 0,Y 594.333,Z 678.449,A -85,B 0,C 180,E1 -954.679,E2 -954.679} C_VEL
LIN {X 0,Y 594.351,Z 678.453,A -85,B 0,C 180,E1 -957.093,E2 -957.093} C_VEL
LIN {X 0,Y 594.357,Z 678.446,A -85,B 0,C 180,E1 -959.677,E2 -959.677} C_VEL
LIN {X 0,Y 594.348,Z 678.445,A -85,B 0,C 180,E1 -962.535,E2 -962.535} C_VEL
LIN {X 0,Y 594.341,Z 678.451,A -85,B 0,C 180,E1 -965.577,E2 -965.577} C_VEL
LIN {X 0,Y 594.321,Z 678.451,A -85,B 0,C 180,E1 -967.762,E2 -967.762} C_VEL
LIN {X 0,Y 594.342,Z 678.447,A -85,B 0,C 180,E1 -969.942,E2 -969.942} C_VEL
LIN {X 0,Y 594.311,Z 678.45,A -85,B 0,C 180,E1 -972.09,E2 -972.09} C_VEL
LIN {X 0,Y 594.31,Z 678.45,A -85,B 0,C 180,E1 -974.214,E2 -974.214} C_VEL
LIN {X 0,Y 594.355,Z 678.447,A -85,B 0,C 180,E1 -976.97,E2 -976.97} C_VEL
LIN {X 0,Y 594.375,Z 678.753,A -85,B 0,C 180,E1 -977.013,E2 -977.013} C_VEL
LIN {X 0,Y 594.733,Z 682.327,A -85,B 0,C 180,E1 -977.065,E2 -977.065} C_VEL
LIN {X 0,Y 594.618,Z 761.435,A -85,B 0,C 180,E1 -978.037,E2 -978.037} C_VEL
LIN {X 0,Y 594.56,Z 773.442,A -85,B 0,C 180,E1 -978.296,E2 -978.296} C_VEL
LIN {X 0,Y 594.551,Z 786.177,A -85,B 0,C 180,E1 -978.709,E2 -978.709} C_VEL
LIN {X 0,Y 594.537,Z 798.693,A -85,B 0,C 180,E1 -979.266,E2 -979.266} C_VEL
LIN {X 0,Y 594.469,Z 810.434,A -85,B 0,C 180,E1 -979.954,E2 -979.954} C_VEL
LIN {X 0,Y 594.405,Z 819.893,A -85,B 0,C 180,E1 -980.64,E2 -980.64} C_VEL
LIN {X 0,Y 594.379,Z 827.796,A -85,B 0,C 180,E1 -981.325,E2 -981.325} C_VEL
LIN {X 0,Y 594.348,Z 836.022,A -85,B 0,C 180,E1 -982.18,E2 -982.18} C_VEL
LIN {X 0,Y 594.312,Z 842.856,A -85,B 0,C 180,E1 -983.034,E2 -983.034} C_VEL
LIN {X 0,Y 594.305,Z 849.569,A -85,B 0,C 180,E1 -984.057,E2 -984.057} C_VEL
LIN {X 0,Y 594.24,Z 855.733,A -85,B 0,C 180,E1 -985.247,E2 -985.247} C_VEL
LIN {X 0,Y 594.289,Z 859.726,A -85,B 0,C 180,E1 -986.266,E2 -986.266} C_VEL
LIN {X 0,Y 594.225,Z 862.679,A -85,B 0,C 180,E1 -987.284,E2 -987.284} C_VEL
LIN {X 0,Y 594.24,Z 864.103,A -85,B 0,C 180,E1 -987.962,E2 -987.962} C_VEL
LIN {X 0,Y 594.247,Z 865.128,A -85,B 0,C 180,E1 -988.64,E2 -988.64} C_VEL
LIN {X 0,Y 594.24,Z 865.75,A -85,B 0,C 180,E1 -989.318,E2 -989.318} C_VEL
LIN {X 0,Y 594.239,Z 865.818,A -85,B 0,C 180,E1 -990.673,E2 -990.673} C_VEL
LIN {X 0,Y 594.24,Z 864.281,A -85,B 0,C 180,E1 -992.029,E2 -992.029} C_VEL
LIN {X 0,Y 594.226,Z 862.927,A -85,B 0,C 180,E1 -992.707,E2 -992.707} C_VEL
LIN {X 0,Y 594.288,Z 860.058,A -85,B 0,C 180,E1 -993.725,E2 -993.725} C_VEL
LIN {X 0,Y 594.242,Z 856.165,A -85,B 0,C 180,E1 -994.744,E2 -994.744} C_VEL
LIN {X 0,Y 594.299,Z 851.14,A -85,B 0,C 180,E1 -995.764,E2 -995.764} C_VEL
LIN {X 0,Y 594.311,Z 844.81,A -85,B 0,C 180,E1 -996.786,E2 -996.786} C_VEL
LIN {X 0,Y 594.344,Z 836.885,A -85,B 0,C 180,E1 -997.811,E2 -997.811} C_VEL
LIN {X 0,Y 594.364,Z 828.821,A -85,B 0,C 180,E1 -998.666,E2 -998.666} C_VEL
LIN {X 0,Y 594.418,Z 820.058,A -85,B 0,C 180,E1 -999.437,E2 -999.437} C_VEL
LIN {X 0,Y 594.465,Z 809.352,A -85,B 0,C 180,E1 -1000.209,E2 -1000.209} C_VEL
LIN {X 0,Y 594.54,Z 797.212,A -85,B 0,C 180,E1 -1000.897,E2 -1000.897} C_VEL
LIN {X 0,Y 594.523,Z 785.203,A -85,B 0,C 180,E1 -1001.419,E2 -1001.419} C_VEL
LIN {X 0,Y 594.568,Z 773.093,A -85,B 0,C 180,E1 -1001.803,E2 -1001.803} C_VEL
LIN {X 0,Y 594.632,Z 760.89,A -85,B 0,C 180,E1 -1002.061,E2 -1002.061} C_VEL
LIN {X 0,Y 594.662,Z 679.768,A -85,B 0,C 180,E1 -1003.058,E2 -1003.058} C_VEL
LIN {X 0,Y 594.364,Z 678.447,A -85,B 0,C 180,E1 -1003.086,E2 -1003.086} C_VEL
LIN {X 0,Y 594.331,Z 678.446,A -85,B 0,C 180,E1 -1005.776,E2 -1005.776} C_VEL
LIN {X 0,Y 594.318,Z 678.448,A -85,B 0,C 180,E1 -1007.9,E2 -1007.9} C_VEL
LIN {X 0,Y 594.392,Z 678.447,A -85,B 0,C 180,E1 -1010.77,E2 -1010.77} C_VEL
LIN {X 0,Y 594.339,Z 678.446,A -85,B 0,C 180,E1 -1013.7,E2 -1013.7} C_VEL
LIN {X 0,Y 594.363,Z 678.445,A -85,B 0,C 180,E1 -1016.694,E2 -1016.694} C_VEL
LIN {X 0,Y 594.351,Z 678.451,A -85,B 0,C 180,E1 -1018.993,E2 -1018.993} C_VEL
LIN {X 0,Y 594.357,Z 678.447,A -85,B 0,C 180,E1 -1021.639,E2 -1021.639} C_VEL
LIN {X 0,Y 594.357,Z 678.443,A -85,B 0,C 180,E1 -1024.573,E2 -1024.573} C_VEL
LIN {X 0,Y 594.351,Z 678.45,A -85,B 0,C 180,E1 -1027.603,E2 -1027.603} C_VEL
LIN {X 0,Y 594.322,Z 678.447,A -85,B 0,C 180,E1 -1030.562,E2 -1030.562} C_VEL
LIN {X 0,Y 594.332,Z 678.451,A -85,B 0,C 180,E1 -1033.293,E2 -1033.293} C_VEL
LIN {X 0,Y 594.316,Z 678.451,A -85,B 0,C 180,E1 -1036.155,E2 -1036.155} C_VEL
LIN {X 0,Y 594.33,Z 678.446,A -85,B 0,C 180,E1 -1038.532,E2 -1038.532} C_VEL
LIN {X 0,Y 594.339,Z 678.447,A -85,B 0,C 180,E1 -1041.289,E2 -1041.289} C_VEL
LIN {X 0,Y 594.343,Z 678.452,A -85,B 0,C 180,E1 -1043.755,E2 -1043.755} C_VEL
LIN {X 0,Y 594.335,Z 678.452,A -85,B 0,C 180,E1 -1046.236,E2 -1046.236} C_VEL
LIN {X 0,Y 594.33,Z 678.448,A -85,B 0,C 180,E1 -1048.647,E2 -1048.647} C_VEL
LIN {X 0,Y 594.325,Z 678.446,A -85,B 0,C 180,E1 -1051.036,E2 -1051.036} C_VEL
LIN {X 0,Y 594.355,Z 678.451,A -85,B 0,C 180,E1 -1054.055,E2 -1054.055} C_VEL
LIN {X 0,Y 594.299,Z 678.45,A -85,B 0,C 180,E1 -1057.03,E2 -1057.03} C_VEL
LIN {X 0,Y 594.329,Z 678.446,A -85,B 0,C 180,E1 -1059.222,E2 -1059.222} C_VEL
LIN {X 0,Y 594.335,Z 678.449,A -85,B 0,C 180,E1 -1062.094,E2 -1062.094} C_VEL
LIN {X 0,Y 594.318,Z 678.452,A -85,B 0,C 180,E1 -1064.921,E2 -1064.921} C_VEL
LIN {X 0,Y 594.325,Z 678.446,A -85,B 0,C 180,E1 -1067.71,E2 -1067.71} C_VEL
LIN {X 0,Y 594.327,Z 678.445,A -85,B 0,C 180,E1 -1069.783,E2 -1069.783} C_VEL
LIN {X 0,Y 594.355,Z 678.449,A -85,B 0,C 180,E1 -1072.526,E2 -1072.526} C_VEL
LIN {X 0,Y 594.338,Z 678.448,A -85,B 0,C 180,E1 -1075.252,E2 -1075.252} C_VEL
LIN {X 0,Y 594.314,Z 678.448,A -85,B 0,C 180,E1 -1077.967,E2 -1077.967} C_VEL
LIN {X 0,Y 594.366,Z 678.447,A -85,B 0,C 180,E1 -1080.677,E2 -1080.677} C_VEL
LIN {X 0,Y 594.35,Z 678.449,A -85,B 0,C 180,E1 -1083.389,E2 -1083.389} C_VEL
LIN {X 0,Y 594.293,Z 678.451,A -85,B 0,C 180,E1 -1086.11,E2 -1086.11} C_VEL
LIN {X 0,Y 594.344,Z 678.444,A -85,B 0,C 180,E1 -1088.158,E2 -1088.158} C_VEL
LIN {X 0,Y 594.374,Z 678.447,A -85,B 0,C 180,E1 -1091.109,E2 -1091.109} C_VEL
LIN {X 0,Y 594.334,Z 678.446,A -85,B 0,C 180,E1 -1094.187,E2 -1094.187} C_VEL
LIN {X 0,Y 594.335,Z 678.451,A -85,B 0,C 180,E1 -1097.195,E2 -1097.195} C_VEL
LIN {X 0,Y 594.325,Z 678.449,A -85,B 0,C 180,E1 -1100.056,E2 -1100.056} C_VEL
LIN {X 0,Y 594.295,Z 678.45,A -85,B 0,C 180,E1 -1102.74,E2 -1102.74} C_VEL
LIN {X 0,Y 594.336,Z 678.447,A -85,B 0,C 180,E1 -1105.195,E2 -1105.195} C_VEL
LIN {X 0,Y 594.317,Z 678.453,A -85,B 0,C 180,E1 -1107.531,E2 -1107.531} C_VEL
LIN {X 0,Y 594.364,Z 678.445,A -85,B 0,C 180,E1 -1110.34,E2 -1110.34} C_VEL
LIN {X 0,Y 594.321,Z 678.447,A -85,B 0,C 180,E1 -1112.954,E2 -1112.954} C_VEL
LIN {X 0,Y 594.323,Z 678.448,A -85,B 0,C 180,E1 -1115.411,E2 -1115.411} C_VEL
LIN {X 0,Y 594.348,Z 678.451,A -85,B 0,C 180,E1 -1117.944,E2 -1117.944} C_VEL
LIN {X 0,Y 594.339,Z 678.446,A -85,B 0,C 180,E1 -1120.829,E2 -1120.829} C_VEL
LIN {X 0,Y 594.336,Z 678.445,A -85,B 0,C 180,E1 -1123.302,E2 -1123.302} C_VEL
LIN {X 0,Y 594.334,Z 678.453,A -85,B 0,C 180,E1 -1126.164,E2 -1126.164} C_VEL
LIN {X 0,Y 594.339,Z 678.446,A -85,B 0,C 180,E1 -1129.183,E2 -1129.183} C_VEL
LIN {X 0,Y 594.34,Z 678.448,A -85,B 0,C 180,E1 -1132.065,E2 -1132.065} C_VEL
LIN {X 0,Y 594.346,Z 678.454,A -85,B 0,C 180,E1 -1134.678,E2 -1134.678} C_VEL
LIN {X 0,Y 594.343,Z 678.449,A -85,B 0,C 180,E1 -1137.094,E2 -1137.094} C_VEL
LIN {X 0,Y 594.337,Z 678.446,A -85,B 0,C 180,E1 -1139.681,E2 -1139.681} C_VEL
LIN {X 0,Y 594.347,Z 678.451,A -85,B 0,C 180,E1 -1142.545,E2 -1142.545} C_VEL
LIN {X 0,Y 594.366,Z 678.535,A -85,B 0,C 180,E1 -1143.386,E2 -1143.386} C_VEL
LIN {X 0,Y 595.142,Z 683.462,A -85,B 0,C 180,E1 -1143.977,E2 -1143.977} C_VEL
LIN {X 0,Y 595.037,Z 708.086,A -85,B 0,C 180,E1 -1146.699,E2 -1146.699} C_VEL
LIN {X 0,Y 594.854,Z 733.299,A -85,B 0,C 180,E1 -1149.428,E2 -1149.428} C_VEL
LIN {X 0,Y 594.684,Z 758.513,A -85,B 0,C 180,E1 -1152.111,E2 -1152.111} C_VEL
LIN {X 0,Y 594.542,Z 783.726,A -85,B 0,C 180,E1 -1154.757,E2 -1154.757} C_VEL
LIN {X 0,Y 594.467,Z 801.916,A -85,B 0,C 180,E1 -1156.644,E2 -1156.644} C_VEL
LIN {X 0,Y 594.731,Z 815.331,A -85,B 0,C 180,E1 -1156.813,E2 -1156.813} C_VEL
LIN {X 0,Y 594.622,Z 912.233,A -85,B 0,C 180,E1 -1158.003,E2 -1158.003} C_VEL
LIN {X 0,Y 594.603,Z 925.405,A -85,B 0,C 180,E1 -1158.306,E2 -1158.306} C_VEL
LIN {X 0,Y 594.565,Z 937.575,A -85,B 0,C 180,E1 -1158.718,E2 -1158.718} C_VEL
LIN {X 0,Y 594.531,Z 949.732,A -85,B 0,C 180,E1 -1159.275,E2 -1159.275} C_VEL
LIN {X 0,Y 594.459,Z 961.277,A -85,B 0,C 180,E1 -1159.963,E2 -1159.963} C_VEL
LIN {X 0,Y 594.43,Z 971.659,A -85,B 0,C 180,E1 -1160.735,E2 -1160.735} C_VEL
LIN {X 0,Y 594.364,Z 980.069,A -85,B 0,C 180,E1 -1161.505,E2 -1161.505} C_VEL
LIN {X 0,Y 594.344,Z 988.003,A -85,B 0,C 180,E1 -1162.36,E2 -1162.36} C_VEL
LIN {X 0,Y 594.277,Z 995.847,A -85,B 0,C 180,E1 -1163.413,E2 -1163.413} C_VEL
LIN {X 0,Y 594.289,Z 1002.706,A -85,B 0,C 180,E1 -1164.576,E2 -1164.576} C_VEL
LIN {X 0,Y 594.269,Z 1007.391,A -85,B 0,C 180,E1 -1165.596,E2 -1165.596} C_VEL
LIN {X 0,Y 594.267,Z 1010.971,A -85,B 0,C 180,E1 -1166.615,E2 -1166.615} C_VEL
LIN {X 0,Y 594.225,Z 1012.821,A -85,B 0,C 180,E1 -1167.293,E2 -1167.293} C_VEL
LIN {X 0,Y 594.24,Z 1014.21,A -85,B 0,C 180,E1 -1167.971,E2 -1167.971} C_VEL
LIN {X 0,Y 594.239,Z 1015.787,A -85,B 0,C 180,E1 -1169.327,E2 -1169.327} C_VEL
LIN {X 0,Y 594.236,Z 1016,A -85,B 0,C 180,E1 -1170.004,E2 -1170.004} C_VEL
LIN {X 0,Y 594.247,Z 1015.179,A -85,B 0,C 180,E1 -1171.36,E2 -1171.36} C_VEL
LIN {X 0,Y 594.24,Z 1014.195,A -85,B 0,C 180,E1 -1172.038,E2 -1172.038} C_VEL
LIN {X 0,Y 594.226,Z 1012.798,A -85,B 0,C 180,E1 -1172.716,E2 -1172.716} C_VEL
LIN {X 0,Y 594.289,Z 1009.882,A -85,B 0,C 180,E1 -1173.734,E2 -1173.734} C_VEL
LIN {X 0,Y 594.241,Z 1005.932,A -85,B 0,C 180,E1 -1174.753,E2 -1174.753} C_VEL
LIN {X 0,Y 594.305,Z 999.853,A -85,B 0,C 180,E1 -1175.943,E2 -1175.943} C_VEL
LIN {X 0,Y 594.312,Z 993.206,A -85,B 0,C 180,E1 -1176.966,E2 -1176.966} C_VEL
LIN {X 0,Y 594.361,Z 984.955,A -85,B 0,C 180,E1 -1177.99,E2 -1177.99} C_VEL
LIN {X 0,Y 594.406,Z 974.555,A -85,B 0,C 180,E1 -1179.017,E2 -1179.017} C_VEL
LIN {X 0,Y 594.449,Z 963.692,A -85,B 0,C 180,E1 -1179.875,E2 -1179.875} C_VEL
LIN {X 0,Y 594.506,Z 952.705,A -85,B 0,C 180,E1 -1180.562,E2 -1180.562} C_VEL
LIN {X 0,Y 594.559,Z 940.061,A -85,B 0,C 180,E1 -1181.18,E2 -1181.18} C_VEL
LIN {X 0,Y 594.579,Z 928.765,A -85,B 0,C 180,E1 -1181.596,E2 -1181.596} C_VEL
LIN {X 0,Y 594.614,Z 916.314,A -85,B 0,C 180,E1 -1181.919,E2 -1181.919} C_VEL
LIN {X 0,Y 594.654,Z 900.423,A -85,B 0,C 180,E1 -1182.157,E2 -1182.157} C_VEL
LIN {X 0,Y 594.589,Z 802.722,A -85,B 0,C 180,E1 -1183.343,E2 -1183.343} C_VEL
LIN {X 0,Y 594.467,Z 801.706,A -85,B 0,C 180,E1 -1183.376,E2 -1183.376} C_VEL
LIN {X 0,Y 594.602,Z 775.232,A -85,B 0,C 180,E1 -1186.13,E2 -1186.13} C_VEL
LIN {X 0,Y 594.769,Z 746.957,A -85,B 0,C 180,E1 -1189.113,E2 -1189.113} C_VEL
LIN {X 0,Y 594.954,Z 721.444,A -85,B 0,C 180,E1 -1191.848,E2 -1191.848} C_VEL
LIN {X 0,Y 595.084,Z 696.452,A -85,B 0,C 180,E1 -1194.58,E2 -1194.58} C_VEL
LIN {X 0,Y 595.158,Z 682.113,A -85,B 0,C 180,E1 -1196.174,E2 -1196.174} C_VEL
LIN {X 0,Y 594.363,Z 678.451,A -85,B 0,C 180,E1 -1196.643,E2 -1196.643} C_VEL
LIN {X 0,Y 594.318,Z 678.45,A -85,B 0,C 180,E1 -1199.782,E2 -1199.782} C_VEL
LIN {X 0,Y 594.334,Z 678.446,A -85,B 0,C 180,E1 -1202.152,E2 -1202.152} C_VEL
LIN {X 0,Y 594.303,Z 678.452,A -85,B 0,C 180,E1 -1204.588,E2 -1204.588} C_VEL
LIN {X 0,Y 594.338,Z 678.455,A -85,B 0,C 180,E1 -1207.093,E2 -1207.093} C_VEL
LIN {X 0,Y 594.332,Z 678.448,A -85,B 0,C 180,E1 -1209.769,E2 -1209.769} C_VEL
LIN {X 0,Y 594.327,Z 678.447,A -85,B 0,C 180,E1 -1212.382,E2 -1212.382} C_VEL
LIN {X 0,Y 594.34,Z 678.456,A -85,B 0,C 180,E1 -1215.196,E2 -1215.196} C_VEL
LIN {X 0,Y 594.369,Z 678.441,A -85,B 0,C 180,E1 -1218.155,E2 -1218.155} C_VEL
LIN {X 0,Y 594.371,Z 678.451,A -85,B 0,C 180,E1 -1221.194,E2 -1221.194} C_VEL
LIN {X 0,Y 594.355,Z 678.446,A -85,B 0,C 180,E1 -1223.756,E2 -1223.756} C_VEL
LIN {X 0,Y 594.363,Z 678.442,A -85,B 0,C 180,E1 -1226.238,E2 -1226.238} C_VEL
LIN {X 0,Y 594.37,Z 678.443,A -85,B 0,C 180,E1 -1228.65,E2 -1228.65} C_VEL
LIN {X 0,Y 594.387,Z 678.445,A -85,B 0,C 180,E1 -1231.044,E2 -1231.044} C_VEL
LIN {X 0,Y 594.373,Z 678.442,A -85,B 0,C 180,E1 -1234.056,E2 -1234.056} C_VEL
LIN {X 0,Y 594.378,Z 678.44,A -85,B 0,C 180,E1 -1236.295,E2 -1236.295} C_VEL
LIN {X 0,Y 594.407,Z 678.445,A -85,B 0,C 180,E1 -1239.224,E2 -1239.224} C_VEL
LIN {X 0,Y 594.352,Z 678.445,A -85,B 0,C 180,E1 -1242.095,E2 -1242.095} C_VEL
LIN {X 0,Y 594.363,Z 678.443,A -85,B 0,C 180,E1 -1244.219,E2 -1244.219} C_VEL
LIN {X 0,Y 594.405,Z 678.442,A -85,B 0,C 180,E1 -1247.007,E2 -1247.007} C_VEL
LIN {X 0,Y 594.749,Z 682.629,A -85,B 0,C 180,E1 -1247.069,E2 -1247.069} C_VEL
LIN {X 0,Y 594.665,Z 761.782,A -85,B 0,C 180,E1 -1248.042,E2 -1248.042} C_VEL
LIN {X 0,Y 594.641,Z 774.39,A -85,B 0,C 180,E1 -1248.323,E2 -1248.323} C_VEL
LIN {X 0,Y 594.575,Z 787.247,A -85,B 0,C 180,E1 -1248.751,E2 -1248.751} C_VEL
LIN {X 0,Y 594.548,Z 798.766,A -85,B 0,C 180,E1 -1249.27,E2 -1249.27} C_VEL
LIN {X 0,Y 594.441,Z 809.214,A -85,B 0,C 180,E1 -1249.871,E2 -1249.871} C_VEL
LIN {X 0,Y 594.403,Z 819.964,A -85,B 0,C 180,E1 -1250.644,E2 -1250.644} C_VEL
LIN {X 0,Y 594.379,Z 827.857,A -85,B 0,C 180,E1 -1251.329,E2 -1251.329} C_VEL
LIN {X 0,Y 594.348,Z 837.569,A -85,B 0,C 180,E1 -1252.355,E2 -1252.355} C_VEL
LIN {X 0,Y 594.302,Z 845.426,A -85,B 0,C 180,E1 -1253.395,E2 -1253.395} C_VEL
LIN {X 0,Y 594.289,Z 852.434,A -85,B 0,C 180,E1 -1254.571,E2 -1254.571} C_VEL
LIN {X 0,Y 594.27,Z 857.172,A -85,B 0,C 180,E1 -1255.591,E2 -1255.591} C_VEL
LIN {X 0,Y 594.268,Z 860.804,A -85,B 0,C 180,E1 -1256.61,E2 -1256.61} C_VEL
LIN {X 0,Y 594.225,Z 862.694,A -85,B 0,C 180,E1 -1257.288,E2 -1257.288} C_VEL
LIN {X 0,Y 594.24,Z 864.131,A -85,B 0,C 180,E1 -1257.967,E2 -1257.967} C_VEL
LIN {X 0,Y 594.24,Z 865.754,A -85,B 0,C 180,E1 -1259.322,E2 -1259.322} C_VEL
LIN {X 0,Y 594.236,Z 865.996,A -85,B 0,C 180,E1 -1260,E2 -1260} C_VEL
LIN {X 0,Y 594.239,Z 865.813,A -85,B 0,C 180,E1 -1260.678,E2 -1260.678} C_VEL
LIN {X 0,Y 594.239,Z 864.277,A -85,B 0,C 180,E1 -1262.033,E2 -1262.033} C_VEL
LIN {X 0,Y 594.226,Z 862.898,A -85,B 0,C 180,E1 -1262.712,E2 -1262.712} C_VEL
LIN {X 0,Y 594.289,Z 860.023,A -85,B 0,C 180,E1 -1263.729,E2 -1263.729} C_VEL
LIN {X 0,Y 594.241,Z 856.126,A -85,B 0,C 180,E1 -1264.749,E2 -1264.749} C_VEL
LIN {X 0,Y 594.299,Z 851.1,A -85,B 0,C 180,E1 -1265.769,E2 -1265.769} C_VEL
LIN {X 0,Y 594.286,Z 844.787,A -85,B 0,C 180,E1 -1266.792,E2 -1266.792} C_VEL
LIN {X 0,Y 594.347,Z 836.866,A -85,B 0,C 180,E1 -1267.816,E2 -1267.816} C_VEL
LIN {X 0,Y 594.369,Z 826.991,A -85,B 0,C 180,E1 -1268.842,E2 -1268.842} C_VEL
LIN {X 0,Y 594.425,Z 816.705,A -85,B 0,C 180,E1 -1269.7,E2 -1269.7} C_VEL
LIN {X 0,Y 594.492,Z 805.089,A -85,B 0,C 180,E1 -1270.472,E2 -1270.472} C_VEL
LIN {X 0,Y 594.57,Z 793.167,A -85,B 0,C 180,E1 -1271.087,E2 -1271.087} C_VEL
LIN {X 0,Y 594.597,Z 781.472,A -85,B 0,C 180,E1 -1271.55,E2 -1271.55} C_VEL
LIN {X 0,Y 594.639,Z 772.777,A -85,B 0,C 180,E1 -1271.81,E2 -1271.81} C_VEL
LIN {X 0,Y 593.955,Z 767.107,A -85,B 0,C 180,E1 -1271.962,E2 -1271.962} C_VEL
LIN {X 0,Y 588.84,Z 750.432,A -85,B 0,C 180,E1 -1272.326,E2 -1272.326} C_VEL
LIN {X 0,Y 587.842,Z 744.684,A -85,B 0,C 180,E1 -1272.415,E2 -1272.415} C_VEL
LIN {X 0,Y 587.762,Z 742.735,A -85,B 0,C 180,E1 -1272.44,E2 -1272.44} C_VEL
LIN {X 0,Y 587.73,Z 680.857,A -85,B 0,C 180,E1 -1273.201,E2 -1273.201} C_VEL
LIN {X 0,Y 587.356,Z 679.319,A -85,B 0,C 180,E1 -1273.229,E2 -1273.229} C_VEL
LIN {X 0,Y 587.32,Z 679.321,A -85,B 0,C 180,E1 -1275.975,E2 -1275.975} C_VEL
LIN {X 0,Y 587.351,Z 679.325,A -85,B 0,C 180,E1 -1278.849,E2 -1278.849} C_VEL
LIN {X 0,Y 587.319,Z 679.319,A -85,B 0,C 180,E1 -1281.775,E2 -1281.775} C_VEL
LIN {X 0,Y 587.356,Z 679.325,A -85,B 0,C 180,E1 -1284.758,E2 -1284.758} C_VEL
LIN {X 0,Y 587.313,Z 679.32,A -85,B 0,C 180,E1 -1287.82,E2 -1287.82} C_VEL
LIN {X 0,Y 587.345,Z 679.321,A -85,B 0,C 180,E1 -1290.509,E2 -1290.509} C_VEL
LIN {X 0,Y 587.337,Z 679.32,A -85,B 0,C 180,E1 -1293.397,E2 -1293.397} C_VEL
LIN {X 0,Y 587.292,Z 679.323,A -85,B 0,C 180,E1 -1295.9,E2 -1295.9} C_VEL
LIN {X 0,Y 587.33,Z 679.321,A -85,B 0,C 180,E1 -1298.48,E2 -1298.48} C_VEL
LIN {X 0,Y 587.322,Z 679.327,A -85,B 0,C 180,E1 -1301.158,E2 -1301.158} C_VEL
LIN {X 0,Y 587.315,Z 679.32,A -85,B 0,C 180,E1 -1304.11,E2 -1304.11} C_VEL
LIN {X 0,Y 587.298,Z 679.331,A -85,B 0,C 180,E1 -1306.99,E2 -1306.99} C_VEL
LIN {X 0,Y 587.304,Z 679.322,A -85,B 0,C 180,E1 -1309.742,E2 -1309.742} C_VEL
LIN {X 0,Y 587.322,Z 679.32,A -85,B 0,C 180,E1 -1312.388,E2 -1312.388} C_VEL
LIN {X 0,Y 587.325,Z 679.321,A -85,B 0,C 180,E1 -1315.656,E2 -1315.656} C_VEL
LIN {X 0,Y 587.313,Z 679.32,A -85,B 0,C 180,E1 -1318.226,E2 -1318.226} C_VEL
LIN {X 0,Y 587.312,Z 679.325,A -85,B 0,C 180,E1 -1320.874,E2 -1320.874} C_VEL
LIN {X 0,Y 587.288,Z 679.326,A -85,B 0,C 180,E1 -1323.834,E2 -1323.834} C_VEL
LIN {X 0,Y 587.294,Z 679.325,A -85,B 0,C 180,E1 -1326.737,E2 -1326.737} C_VEL
LIN {X 0,Y 587.307,Z 679.326,A -85,B 0,C 180,E1 -1329.691,E2 -1329.691} C_VEL
LIN {X 0,Y 587.272,Z 679.329,A -85,B 0,C 180,E1 -1331.868,E2 -1331.868} C_VEL
LIN {X 0,Y 587.278,Z 679.327,A -85,B 0,C 180,E1 -1334.02,E2 -1334.02} C_VEL
LIN {X 0,Y 587.317,Z 679.322,A -85,B 0,C 180,E1 -1336.15,E2 -1336.15} C_VEL
LIN {X 0,Y 587.3,Z 679.326,A -85,B 0,C 180,E1 -1336.854,E2 -1336.854} C_VEL
LIN {X 0,Y 587.814,Z 682.372,A -85,B 0,C 180,E1 -1336.91,E2 -1336.91} C_VEL
LIN {X 0,Y 587.678,Z 761.39,A -85,B 0,C 180,E1 -1337.894,E2 -1337.894} C_VEL
LIN {X 0,Y 587.622,Z 772.567,A -85,B 0,C 180,E1 -1338.134,E2 -1338.134} C_VEL
LIN {X 0,Y 587.587,Z 784.186,A -85,B 0,C 180,E1 -1338.499,E2 -1338.499} C_VEL
LIN {X 0,Y 587.552,Z 796.967,A -85,B 0,C 180,E1 -1339.05,E2 -1339.05} C_VEL
LIN {X 0,Y 587.438,Z 809.152,A -85,B 0,C 180,E1 -1339.745,E2 -1339.745} C_VEL
LIN {X 0,Y 587.393,Z 818.828,A -85,B 0,C 180,E1 -1340.44,E2 -1340.44} C_VEL
LIN {X 0,Y 587.34,Z 827.789,A -85,B 0,C 180,E1 -1341.22,E2 -1341.22} C_VEL
LIN {X 0,Y 587.29,Z 836.015,A -85,B 0,C 180,E1 -1342.086,E2 -1342.086} C_VEL
LIN {X 0,Y 587.25,Z 842.849,A -85,B 0,C 180,E1 -1342.95,E2 -1342.95} C_VEL
LIN {X 0,Y 587.218,Z 849.565,A -85,B 0,C 180,E1 -1343.985,E2 -1343.985} C_VEL
LIN {X 0,Y 587.167,Z 854.111,A -85,B 0,C 180,E1 -1344.845,E2 -1344.845} C_VEL
LIN {X 0,Y 587.182,Z 858.481,A -85,B 0,C 180,E1 -1345.878,E2 -1345.878} C_VEL
LIN {X 0,Y 587.194,Z 860.81,A -85,B 0,C 180,E1 -1346.565,E2 -1346.565} C_VEL
LIN {X 0,Y 587.132,Z 862.68,A -85,B 0,C 180,E1 -1347.251,E2 -1347.251} C_VEL
LIN {X 0,Y 587.146,Z 865.129,A -85,B 0,C 180,E1 -1348.624,E2 -1348.624} C_VEL
LIN {X 0,Y 587.14,Z 865.75,A -85,B 0,C 180,E1 -1349.31,E2 -1349.31} C_VEL
LIN {X 0,Y 587.14,Z 865.818,A -85,B 0,C 180,E1 -1350.681,E2 -1350.681} C_VEL
LIN {X 0,Y 587.147,Z 865.242,A -85,B 0,C 180,E1 -1351.367,E2 -1351.367} C_VEL
LIN {X 0,Y 587.132,Z 862.926,A -85,B 0,C 180,E1 -1352.74,E2 -1352.74} C_VEL
LIN {X 0,Y 587.212,Z 860.058,A -85,B 0,C 180,E1 -1353.769,E2 -1353.769} C_VEL
LIN {X 0,Y 587.147,Z 856.165,A -85,B 0,C 180,E1 -1354.801,E2 -1354.801} C_VEL
LIN {X 0,Y 587.209,Z 850.147,A -85,B 0,C 180,E1 -1356.006,E2 -1356.006} C_VEL
LIN {X 0,Y 587.24,Z 843.56,A -85,B 0,C 180,E1 -1357.041,E2 -1357.041} C_VEL
LIN {X 0,Y 587.271,Z 836.869,A -85,B 0,C 180,E1 -1357.905,E2 -1357.905} C_VEL
LIN {X 0,Y 587.322,Z 828.804,A -85,B 0,C 180,E1 -1358.771,E2 -1358.771} C_VEL
LIN {X 0,Y 587.389,Z 820.038,A -85,B 0,C 180,E1 -1359.551,E2 -1359.551} C_VEL
LIN {X 0,Y 587.439,Z 810.608,A -85,B 0,C 180,E1 -1360.246,E2 -1360.246} C_VEL
LIN {X 0,Y 587.559,Z 798.929,A -85,B 0,C 180,E1 -1360.941,E2 -1360.941} C_VEL
LIN {X 0,Y 587.548,Z 785.506,A -85,B 0,C 180,E1 -1361.545,E2 -1361.545} C_VEL
LIN {X 0,Y 587.611,Z 773.022,A -85,B 0,C 180,E1 -1361.945,E2 -1361.945} C_VEL
LIN {X 0,Y 587.675,Z 762.09,A -85,B 0,C 180,E1 -1362.184,E2 -1362.184} C_VEL
LIN {X 0,Y 587.723,Z 680.951,A -85,B 0,C 180,E1 -1363.2,E2 -1363.2} C_VEL
LIN {X 0,Y 587.335,Z 679.321,A -85,B 0,C 180,E1 -1363.246,E2 -1363.246} C_VEL
LIN {X 0,Y 587.294,Z 679.324,A -85,B 0,C 180,E1 -1365.97,E2 -1365.97} C_VEL
LIN {X 0,Y 587.335,Z 679.329,A -85,B 0,C 180,E1 -1368.843,E2 -1368.843} C_VEL
LIN {X 0,Y 587.29,Z 679.323,A -85,B 0,C 180,E1 -1371.769,E2 -1371.769} C_VEL
LIN {X 0,Y 587.29,Z 679.328,A -85,B 0,C 180,E1 -1374.754,E2 -1374.754} C_VEL
LIN {X 0,Y 587.324,Z 679.321,A -85,B 0,C 180,E1 -1377.687,E2 -1377.687} C_VEL
LIN {X 0,Y 587.297,Z 679.323,A -85,B 0,C 180,E1 -1380.503,E2 -1380.503} C_VEL
LIN {X 0,Y 587.305,Z 679.328,A -85,B 0,C 180,E1 -1383.106,E2 -1383.106} C_VEL
LIN {X 0,Y 587.306,Z 679.329,A -85,B 0,C 180,E1 -1385.538,E2 -1385.538} C_VEL
LIN {X 0,Y 587.283,Z 679.322,A -85,B 0,C 180,E1 -1388.474,E2 -1388.474} C_VEL
LIN {X 0,Y 587.322,Z 679.323,A -85,B 0,C 180,E1 -1391.149,E2 -1391.149} C_VEL
LIN {X 0,Y 587.285,Z 679.325,A -85,B 0,C 180,E1 -1394.109,E2 -1394.109} C_VEL
LIN {X 0,Y 587.285,Z 679.324,A -85,B 0,C 180,E1 -1396.991,E2 -1396.991} C_VEL
LIN {X 0,Y 587.303,Z 679.329,A -85,B 0,C 180,E1 -1399.972,E2 -1399.972} C_VEL
LIN {X 0,Y 587.293,Z 679.325,A -85,B 0,C 180,E1 -1402.388,E2 -1402.388} C_VEL
LIN {X 0,Y 587.289,Z 679.323,A -85,B 0,C 180,E1 -1404.942,E2 -1404.942} C_VEL
LIN {X 0,Y 587.284,Z 679.325,A -85,B 0,C 180,E1 -1407.417,E2 -1407.417} C_VEL
LIN {X 0,Y 587.312,Z 679.326,A -85,B 0,C 180,E1 -1409.828,E2 -1409.828} C_VEL
LIN {X 0,Y 587.274,Z 679.325,A -85,B 0,C 180,E1 -1412.951,E2 -1412.951} C_VEL
LIN {X 0,Y 587.288,Z 679.323,A -85,B 0,C 180,E1 -1415.414,E2 -1415.414} C_VEL
LIN {X 0,Y 587.27,Z 679.334,A -85,B 0,C 180,E1 -1418.224,E2 -1418.224} C_VEL
LIN {X 0,Y 587.278,Z 679.325,A -85,B 0,C 180,E1 -1421.149,E2 -1421.149} C_VEL
LIN {X 0,Y 587.277,Z 679.324,A -85,B 0,C 180,E1 -1423.309,E2 -1423.309} C_VEL
LIN {X 0,Y 587.303,Z 679.325,A -85,B 0,C 180,E1 -1426.153,E2 -1426.153} C_VEL
LIN {X 0,Y 587.331,Z 679.323,A -85,B 0,C 180,E1 -1428.962,E2 -1428.962} C_VEL
LIN {X 0,Y 587.298,Z 679.322,A -85,B 0,C 180,E1 -1431.744,E2 -1431.744} C_VEL
LIN {X 0,Y 587.327,Z 679.324,A -85,B 0,C 180,E1 -1434.507,E2 -1434.507} C_VEL
LIN {X 0,Y 587.316,Z 679.325,A -85,B 0,C 180,E1 -1437.256,E2 -1437.256} C_VEL
LIN {X 0,Y 587.298,Z 679.322,A -85,B 0,C 180,E1 -1440,E2 -1440} C_VEL
LIN {X 0,Y 587.316,Z 679.324,A -85,B 0,C 180,E1 -1442.743,E2 -1442.743} C_VEL
LIN {X 0,Y 587.328,Z 679.324,A -85,B 0,C 180,E1 -1445.493,E2 -1445.493} C_VEL
LIN {X 0,Y 587.298,Z 679.321,A -85,B 0,C 180,E1 -1448.256,E2 -1448.256} C_VEL
LIN {X 0,Y 587.33,Z 679.326,A -85,B 0,C 180,E1 -1451.167,E2 -1451.167} C_VEL
LIN {X 0,Y 587.303,Z 679.321,A -85,B 0,C 180,E1 -1454.27,E2 -1454.27} C_VEL
LIN {X 0,Y 587.302,Z 679.331,A -85,B 0,C 180,E1 -1457.407,E2 -1457.407} C_VEL
LIN {X 0,Y 587.271,Z 679.325,A -85,B 0,C 180,E1 -1460.307,E2 -1460.307} C_VEL
LIN {X 0,Y 587.252,Z 679.328,A -85,B 0,C 180,E1 -1462.874,E2 -1462.874} C_VEL
LIN {X 0,Y 587.301,Z 679.328,A -85,B 0,C 180,E1 -1465.518,E2 -1465.518} C_VEL
LIN {X 0,Y 587.283,Z 679.335,A -85,B 0,C 180,E1 -1467.821,E2 -1467.821} C_VEL
LIN {X 0,Y 587.305,Z 679.322,A -85,B 0,C 180,E1 -1470.52,E2 -1470.52} C_VEL
LIN {X 0,Y 587.282,Z 679.326,A -85,B 0,C 180,E1 -1473.4,E2 -1473.4} C_VEL
LIN {X 0,Y 587.3,Z 679.33,A -85,B 0,C 180,E1 -1475.9,E2 -1475.9} C_VEL
LIN {X 0,Y 587.286,Z 679.327,A -85,B 0,C 180,E1 -1478.483,E2 -1478.483} C_VEL
LIN {X 0,Y 587.308,Z 679.321,A -85,B 0,C 180,E1 -1481.16,E2 -1481.16} C_VEL
LIN {X 0,Y 587.282,Z 679.332,A -85,B 0,C 180,E1 -1484.119,E2 -1484.119} C_VEL
LIN {X 0,Y 587.272,Z 679.326,A -85,B 0,C 180,E1 -1487,E2 -1487} C_VEL
LIN {X 0,Y 587.274,Z 679.326,A -85,B 0,C 180,E1 -1489.752,E2 -1489.752} C_VEL
LIN {X 0,Y 587.307,Z 679.329,A -85,B 0,C 180,E1 -1492.398,E2 -1492.398} C_VEL
LIN {X 0,Y 587.311,Z 679.325,A -85,B 0,C 180,E1 -1494.952,E2 -1494.952} C_VEL
LIN {X 0,Y 587.301,Z 679.323,A -85,B 0,C 180,E1 -1497.427,E2 -1497.427} C_VEL
LIN {X 0,Y 587.285,Z 679.325,A -85,B 0,C 180,E1 -1499.835,E2 -1499.835} C_VEL
LIN {X 0,Y 587.323,Z 679.324,A -85,B 0,C 180,E1 -1502.313,E2 -1502.313} C_VEL
LIN {X 0,Y 587.344,Z 679.512,A -85,B 0,C 180,E1 -1503.154,E2 -1503.154} C_VEL
LIN {X 0,Y 588.39,Z 684.553,A -85,B 0,C 180,E1 -1503.779,E2 -1503.779} C_VEL
LIN {X 0,Y 588.202,Z 709.767,A -85,B 0,C 180,E1 -1506.598,E2 -1506.598} C_VEL
LIN {X 0,Y 587.961,Z 734.98,A -85,B 0,C 180,E1 -1509.359,E2 -1509.359} C_VEL
LIN {X 0,Y 587.768,Z 760.194,A -85,B 0,C 180,E1 -1512.074,E2 -1512.074} C_VEL
LIN {X 0,Y 587.563,Z 785.407,A -85,B 0,C 180,E1 -1514.749,E2 -1514.749} C_VEL
LIN {X 0,Y 587.446,Z 801.915,A -85,B 0,C 180,E1 -1516.482,E2 -1516.482} C_VEL
LIN {X 0,Y 587.827,Z 808.176,A -85,B 0,C 180,E1 -1516.568,E2 -1516.568} C_VEL
LIN {X 0,Y 587.699,Z 912.233,A -85,B 0,C 180,E1 -1517.86,E2 -1517.86} C_VEL
LIN {X 0,Y 587.653,Z 925.405,A -85,B 0,C 180,E1 -1518.166,E2 -1518.166} C_VEL
LIN {X 0,Y 587.594,Z 937.703,A -85,B 0,C 180,E1 -1518.588,E2 -1518.588} C_VEL
LIN {X 0,Y 587.537,Z 949.731,A -85,B 0,C 180,E1 -1519.146,E2 -1519.146} C_VEL
LIN {X 0,Y 587.441,Z 961.278,A -85,B 0,C 180,E1 -1519.841,E2 -1519.841} C_VEL
LIN {X 0,Y 587.408,Z 971.66,A -85,B 0,C 180,E1 -1520.623,E2 -1520.623} C_VEL
LIN {X 0,Y 587.307,Z 980.078,A -85,B 0,C 180,E1 -1521.403,E2 -1521.403} C_VEL
LIN {X 0,Y 587.271,Z 988.003,A -85,B 0,C 180,E1 -1522.268,E2 -1522.268} C_VEL
LIN {X 0,Y 587.229,Z 994.506,A -85,B 0,C 180,E1 -1523.131,E2 -1523.131} C_VEL
LIN {X 0,Y 587.229,Z 1000.893,A -85,B 0,C 180,E1 -1524.166,E2 -1524.166} C_VEL
LIN {X 0,Y 587.147,Z 1005.97,A -85,B 0,C 180,E1 -1525.199,E2 -1525.199} C_VEL
LIN {X 0,Y 587.212,Z 1009.911,A -85,B 0,C 180,E1 -1526.231,E2 -1526.231} C_VEL
LIN {X 0,Y 587.132,Z 1012.821,A -85,B 0,C 180,E1 -1527.26,E2 -1527.26} C_VEL
LIN {X 0,Y 587.139,Z 1014.209,A -85,B 0,C 180,E1 -1527.947,E2 -1527.947} C_VEL
LIN {X 0,Y 587.14,Z 1015.787,A -85,B 0,C 180,E1 -1529.319,E2 -1529.319} C_VEL
LIN {X 0,Y 587.137,Z 1016,A -85,B 0,C 180,E1 -1530.005,E2 -1530.005} C_VEL
LIN {X 0,Y 587.147,Z 1015.18,A -85,B 0,C 180,E1 -1531.376,E2 -1531.376} C_VEL
LIN {X 0,Y 587.139,Z 1014.194,A -85,B 0,C 180,E1 -1532.062,E2 -1532.062} C_VEL
LIN {X 0,Y 587.132,Z 1012.798,A -85,B 0,C 180,E1 -1532.749,E2 -1532.749} C_VEL
LIN {X 0,Y 587.213,Z 1009.882,A -85,B 0,C 180,E1 -1533.779,E2 -1533.779} C_VEL
LIN {X 0,Y 587.147,Z 1005.932,A -85,B 0,C 180,E1 -1534.811,E2 -1534.811} C_VEL
LIN {X 0,Y 587.218,Z 999.853,A -85,B 0,C 180,E1 -1536.015,E2 -1536.015} C_VEL
LIN {X 0,Y 587.249,Z 993.207,A -85,B 0,C 180,E1 -1537.05,E2 -1537.05} C_VEL
LIN {X 0,Y 587.3,Z 984.955,A -85,B 0,C 180,E1 -1538.087,E2 -1538.087} C_VEL
LIN {X 0,Y 587.359,Z 974.556,A -85,B 0,C 180,E1 -1539.126,E2 -1539.126} C_VEL
LIN {X 0,Y 587.433,Z 964.878,A -85,B 0,C 180,E1 -1539.907,E2 -1539.907} C_VEL
LIN {X 0,Y 587.519,Z 954.261,A -85,B 0,C 180,E1 -1540.602,E2 -1540.602} C_VEL
LIN {X 0,Y 587.577,Z 941.652,A -85,B 0,C 180,E1 -1541.244,E2 -1541.244} C_VEL
LIN {X 0,Y 587.601,Z 930.13,A -85,B 0,C 180,E1 -1541.69,E2 -1541.69} C_VEL
LIN {X 0,Y 587.657,Z 917.362,A -85,B 0,C 180,E1 -1542.041,E2 -1542.041} C_VEL
LIN {X 0,Y 587.711,Z 904,A -85,B 0,C 180,E1 -1542.259,E2 -1542.259} C_VEL
LIN {X 0,Y 587.735,Z 803.84,A -85,B 0,C 180,E1 -1543.488,E2 -1543.488} C_VEL
LIN {X 0,Y 587.457,Z 801.706,A -85,B 0,C 180,E1 -1543.538,E2 -1543.538} C_VEL
LIN {X 0,Y 587.664,Z 775.232,A -85,B 0,C 180,E1 -1546.326,E2 -1546.326} C_VEL
LIN {X 0,Y 587.866,Z 747.32,A -85,B 0,C 180,E1 -1549.307,E2 -1549.307} C_VEL
LIN {X 0,Y 588.102,Z 721.444,A -85,B 0,C 180,E1 -1552.116,E2 -1552.116} C_VEL
LIN {X 0,Y 588.31,Z 696.4,A -85,B 0,C 180,E1 -1554.888,E2 -1554.888} C_VEL
LIN {X 0,Y 588.275,Z 683.368,A -85,B 0,C 180,E1 -1556.361,E2 -1556.361} C_VEL
LIN {X 0,Y 587.322,Z 679.33,A -85,B 0,C 180,E1 -1556.881,E2 -1556.881} C_VEL
LIN {X 0,Y 587.291,Z 679.33,A -85,B 0,C 180,E1 -1559.386,E2 -1559.386} C_VEL
LIN {X 0,Y 587.307,Z 679.322,A -85,B 0,C 180,E1 -1561.829,E2 -1561.829} C_VEL
LIN {X 0,Y 587.275,Z 679.326,A -85,B 0,C 180,E1 -1564.337,E2 -1564.337} C_VEL
LIN {X 0,Y 587.312,Z 679.324,A -85,B 0,C 180,E1 -1566.752,E2 -1566.752} C_VEL
LIN {X 0,Y 587.308,Z 679.329,A -85,B 0,C 180,E1 -1569.365,E2 -1569.365} C_VEL
LIN {X 0,Y 587.297,Z 679.323,A -85,B 0,C 180,E1 -1572.103,E2 -1572.103} C_VEL
LIN {X 0,Y 587.289,Z 679.332,A -85,B 0,C 180,E1 -1575.086,E2 -1575.086} C_VEL
LIN {X 0,Y 587.312,Z 679.322,A -85,B 0,C 180,E1 -1577.924,E2 -1577.924} C_VEL
LIN {X 0,Y 587.327,Z 679.32,A -85,B 0,C 180,E1 -1580.639,E2 -1580.639} C_VEL
LIN {X 0,Y 587.324,Z 679.33,A -85,B 0,C 180,E1 -1583.298,E2 -1583.298} C_VEL
LIN {X 0,Y 587.337,Z 679.32,A -85,B 0,C 180,E1 -1585.778,E2 -1585.778} C_VEL
LIN {X 0,Y 587.342,Z 679.317,A -85,B 0,C 180,E1 -1588.231,E2 -1588.231} C_VEL
LIN {X 0,Y 587.353,Z 679.319,A -85,B 0,C 180,E1 -1590.868,E2 -1590.868} C_VEL
LIN {X 0,Y 587.316,Z 679.323,A -85,B 0,C 180,E1 -1593.83,E2 -1593.83} C_VEL
LIN {X 0,Y 587.325,Z 679.321,A -85,B 0,C 180,E1 -1595.993,E2 -1595.993} C_VEL
LIN {X 0,Y 587.323,Z 679.32,A -85,B 0,C 180,E1 -1598.226,E2 -1598.226} C_VEL
LIN {X 0,Y 587.355,Z 679.323,A -85,B 0,C 180,E1 -1601.151,E2 -1601.151} C_VEL
LIN {X 0,Y 587.32,Z 679.322,A -85,B 0,C 180,E1 -1604.025,E2 -1604.025} C_VEL
LIN {X 0,Y 587.357,Z 679.319,A -85,B 0,C 180,E1 -1606.859,E2 -1606.859} C_VEL
LIN {X 0,Y 587.813,Z 681.06,A -85,B 0,C 180,E1 -1606.894,E2 -1606.894} C_VEL
LIN {X 0,Y 587.72,Z 761.787,A -85,B 0,C 180,E1 -1607.899,E2 -1607.899} C_VEL
LIN {X 0,Y 587.691,Z 774.392,A -85,B 0,C 180,E1 -1608.183,E2 -1608.183} C_VEL
LIN {X 0,Y 587.621,Z 786.698,A -85,B 0,C 180,E1 -1608.594,E2 -1608.594} C_VEL
LIN {X 0,Y 587.563,Z 798.777,A -85,B 0,C 180,E1 -1609.141,E2 -1609.141} C_VEL
LIN {X 0,Y 587.432,Z 809.21,A -85,B 0,C 180,E1 -1609.749,E2 -1609.749} C_VEL
LIN {X 0,Y 587.39,Z 818.882,A -85,B 0,C 180,E1 -1610.444,E2 -1610.444} C_VEL
LIN {X 0,Y 587.339,Z 827.851,A -85,B 0,C 180,E1 -1611.224,E2 -1611.224} C_VEL
LIN {X 0,Y 587.289,Z 836.083,A -85,B 0,C 180,E1 -1612.09,E2 -1612.09} C_VEL
LIN {X 0,Y 587.233,Z 844.147,A -85,B 0,C 180,E1 -1613.126,E2 -1613.126} C_VEL
LIN {X 0,Y 587.237,Z 850.617,A -85,B 0,C 180,E1 -1614.161,E2 -1614.161} C_VEL
LIN {X 0,Y 587.146,Z 855.749,A -85,B 0,C 180,E1 -1615.194,E2 -1615.194} C_VEL
LIN {X 0,Y 587.213,Z 859.735,A -85,B 0,C 180,E1 -1616.226,E2 -1616.226} C_VEL
LIN {X 0,Y 587.132,Z 862.691,A -85,B 0,C 180,E1 -1617.256,E2 -1617.256} C_VEL
LIN {X 0,Y 587.139,Z 864.132,A -85,B 0,C 180,E1 -1617.942,E2 -1617.942} C_VEL
LIN {X 0,Y 587.14,Z 865.755,A -85,B 0,C 180,E1 -1619.314,E2 -1619.314} C_VEL
LIN {X 0,Y 587.137,Z 865.996,A -85,B 0,C 180,E1 -1620,E2 -1620} C_VEL
LIN {X 0,Y 587.148,Z 865.232,A -85,B 0,C 180,E1 -1621.372,E2 -1621.372} C_VEL
LIN {X 0,Y 587.138,Z 864.277,A -85,B 0,C 180,E1 -1622.058,E2 -1622.058} C_VEL
LIN {X 0,Y 587.133,Z 862.889,A -85,B 0,C 180,E1 -1622.744,E2 -1622.744} C_VEL
LIN {X 0,Y 587.213,Z 860.014,A -85,B 0,C 180,E1 -1623.774,E2 -1623.774} C_VEL
LIN {X 0,Y 587.147,Z 856.119,A -85,B 0,C 180,E1 -1624.806,E2 -1624.806} C_VEL
LIN {X 0,Y 587.229,Z 851.094,A -85,B 0,C 180,E1 -1625.839,E2 -1625.839} C_VEL
LIN {X 0,Y 587.225,Z 843.558,A -85,B 0,C 180,E1 -1627.046,E2 -1627.046} C_VEL
LIN {X 0,Y 587.287,Z 835.36,A -85,B 0,C 180,E1 -1628.083,E2 -1628.083} C_VEL
LIN {X 0,Y 587.358,Z 825.105,A -85,B 0,C 180,E1 -1629.122,E2 -1629.122} C_VEL
LIN {X 0,Y 587.433,Z 814.369,A -85,B 0,C 180,E1 -1629.99,E2 -1629.99} C_VEL
LIN {X 0,Y 587.498,Z 803.53,A -85,B 0,C 180,E1 -1630.686,E2 -1630.686} C_VEL
LIN {X 0,Y 587.59,Z 792.51,A -85,B 0,C 180,E1 -1631.249,E2 -1631.249} C_VEL
LIN {X 0,Y 587.638,Z 780.191,A -85,B 0,C 180,E1 -1631.731,E2 -1631.731} C_VEL
LIN {X 0,Y 587.689,Z 766.558,A -85,B 0,C 180,E1 -1632.102,E2 -1632.102} C_VEL
LIN {X 0,Y 587.735,Z 752.608,A -85,B 0,C 180,E1 -1632.32,E2 -1632.32} C_VEL
LIN {X 0,Y 587.762,Z 742.735,A -85,B 0,C 180,E1 -1632.44,E2 -1632.44} C_VEL
LIN {X 0,Y 587.12,Z 736.927,A -85,B 0,C 180,E1 -1632.526,E2 -1632.526} C_VEL
LIN {X 0,Y 581.545,Z 718.233,A -85,B 0,C 180,E1 -1632.879,E2 -1632.879} C_VEL
LIN {X 0,Y 580.878,Z 712.426,A -85,B 0,C 180,E1 -1632.966,E2 -1632.966} C_VEL
LIN {X 0,Y 580.925,Z 682.792,A -85,B 0,C 180,E1 -1633.334,E2 -1633.334} C_VEL
LIN {X 0,Y 580.327,Z 680.194,A -85,B 0,C 180,E1 -1633.392,E2 -1633.392} C_VEL
LIN {X 0,Y 580.276,Z 680.2,A -85,B 0,C 180,E1 -1636.175,E2 -1636.175} C_VEL
LIN {X 0,Y 580.306,Z 680.197,A -85,B 0,C 180,E1 -1639.15,E2 -1639.15} C_VEL
LIN {X 0,Y 580.265,Z 680.199,A -85,B 0,C 180,E1 -1642.053,E2 -1642.053} C_VEL
LIN {X 0,Y 580.31,Z 680.199,A -85,B 0,C 180,E1 -1645.08,E2 -1645.08} C_VEL
LIN {X 0,Y 580.288,Z 680.196,A -85,B 0,C 180,E1 -1648.186,E2 -1648.186} C_VEL
LIN {X 0,Y 580.292,Z 680.202,A -85,B 0,C 180,E1 -1650.693,E2 -1650.693} C_VEL
LIN {X 0,Y 580.293,Z 680.199,A -85,B 0,C 180,E1 -1653.312,E2 -1653.312} C_VEL
LIN {X 0,Y 580.243,Z 680.201,A -85,B 0,C 180,E1 -1655.753,E2 -1655.753} C_VEL
LIN {X 0,Y 580.295,Z 680.195,A -85,B 0,C 180,E1 -1658.146,E2 -1658.146} C_VEL
LIN {X 0,Y 580.304,Z 680.201,A -85,B 0,C 180,E1 -1660.843,E2 -1660.843} C_VEL
LIN {X 0,Y 580.253,Z 680.201,A -85,B 0,C 180,E1 -1663.661,E2 -1663.661} C_VEL
LIN {X 0,Y 580.246,Z 680.204,A -85,B 0,C 180,E1 -1666.613,E2 -1666.613} C_VEL
LIN {X 0,Y 580.289,Z 680.205,A -85,B 0,C 180,E1 -1669.153,E2 -1669.153} C_VEL
LIN {X 0,Y 580.255,Z 680.199,A -85,B 0,C 180,E1 -1671.932,E2 -1671.932} C_VEL
LIN {X 0,Y 580.232,Z 680.203,A -85,B 0,C 180,E1 -1674.449,E2 -1674.449} C_VEL
LIN {X 0,Y 580.248,Z 680.207,A -85,B 0,C 180,E1 -1676.97,E2 -1676.97} C_VEL
LIN {X 0,Y 580.263,Z 680.205,A -85,B 0,C 180,E1 -1679.42,E2 -1679.42} C_VEL
LIN {X 0,Y 580.247,Z 680.2,A -85,B 0,C 180,E1 -1682.152,E2 -1682.152} C_VEL
LIN {X 0,Y 580.234,Z 680.207,A -85,B 0,C 180,E1 -1684.914,E2 -1684.914} C_VEL
LIN {X 0,Y 580.285,Z 680.205,A -85,B 0,C 180,E1 -1687.194,E2 -1687.194} C_VEL
LIN {X 0,Y 580.253,Z 680.201,A -85,B 0,C 180,E1 -1690.172,E2 -1690.172} C_VEL
LIN {X 0,Y 580.28,Z 680.203,A -85,B 0,C 180,E1 -1693.098,E2 -1693.098} C_VEL
LIN {X 0,Y 580.281,Z 680.2,A -85,B 0,C 180,E1 -1695.978,E2 -1695.978} C_VEL
LIN {X 0,Y 580.254,Z 680.202,A -85,B 0,C 180,E1 -1696.703,E2 -1696.703} C_VEL
LIN {X 0,Y 580.923,Z 683.312,A -85,B 0,C 180,E1 -1696.763,E2 -1696.763} C_VEL
LIN {X 0,Y 580.734,Z 761.346,A -85,B 0,C 180,E1 -1697.747,E2 -1697.747} C_VEL
LIN {X 0,Y 580.661,Z 772.539,A -85,B 0,C 180,E1 -1697.989,E2 -1697.989} C_VEL
LIN {X 0,Y 580.618,Z 783.722,A -85,B 0,C 180,E1 -1698.343,E2 -1698.343} C_VEL
LIN {X 0,Y 580.597,Z 795.157,A -85,B 0,C 180,E1 -1698.829,E2 -1698.829} C_VEL
LIN {X 0,Y 580.471,Z 807.824,A -85,B 0,C 180,E1 -1699.532,E2 -1699.532} C_VEL
LIN {X 0,Y 580.374,Z 818.821,A -85,B 0,C 180,E1 -1700.323,E2 -1700.323} C_VEL
LIN {X 0,Y 580.311,Z 827.782,A -85,B 0,C 180,E1 -1701.113,E2 -1701.113} C_VEL
LIN {X 0,Y 580.244,Z 836.009,A -85,B 0,C 180,E1 -1701.989,E2 -1701.989} C_VEL
LIN {X 0,Y 580.189,Z 842.842,A -85,B 0,C 180,E1 -1702.864,E2 -1702.864} C_VEL
LIN {X 0,Y 580.144,Z 848.539,A -85,B 0,C 180,E1 -1703.737,E2 -1703.737} C_VEL
LIN {X 0,Y 580.086,Z 854.102,A -85,B 0,C 180,E1 -1704.782,E2 -1704.782} C_VEL
LIN {X 0,Y 580.106,Z 858.471,A -85,B 0,C 180,E1 -1705.827,E2 -1705.827} C_VEL
LIN {X 0,Y 580.123,Z 860.814,A -85,B 0,C 180,E1 -1706.523,E2 -1706.523} C_VEL
LIN {X 0,Y 580.043,Z 862.68,A -85,B 0,C 180,E1 -1707.218,E2 -1707.218} C_VEL
LIN {X 0,Y 580.046,Z 865.13,A -85,B 0,C 180,E1 -1708.607,E2 -1708.607} C_VEL
LIN {X 0,Y 580.041,Z 865.751,A -85,B 0,C 180,E1 -1709.301,E2 -1709.301} C_VEL
LIN {X 0,Y 580.04,Z 865.817,A -85,B 0,C 180,E1 -1710.69,E2 -1710.69} C_VEL
LIN {X 0,Y 580.047,Z 865.241,A -85,B 0,C 180,E1 -1711.384,E2 -1711.384} C_VEL
LIN {X 0,Y 580.043,Z 862.925,A -85,B 0,C 180,E1 -1712.773,E2 -1712.773} C_VEL
LIN {X 0,Y 580.109,Z 860.058,A -85,B 0,C 180,E1 -1713.816,E2 -1713.816} C_VEL
LIN {X 0,Y 580.054,Z 856.165,A -85,B 0,C 180,E1 -1714.86,E2 -1714.86} C_VEL
LIN {X 0,Y 580.135,Z 850.137,A -85,B 0,C 180,E1 -1716.08,E2 -1716.08} C_VEL
LIN {X 0,Y 580.179,Z 843.546,A -85,B 0,C 180,E1 -1717.127,E2 -1717.127} C_VEL
LIN {X 0,Y 580.228,Z 836.853,A -85,B 0,C 180,E1 -1718.002,E2 -1718.002} C_VEL
LIN {X 0,Y 580.295,Z 828.785,A -85,B 0,C 180,E1 -1718.878,E2 -1718.878} C_VEL
LIN {X 0,Y 580.368,Z 820.017,A -85,B 0,C 180,E1 -1719.667,E2 -1719.667} C_VEL
LIN {X 0,Y 580.449,Z 810.585,A -85,B 0,C 180,E1 -1720.37,E2 -1720.37} C_VEL
LIN {X 0,Y 580.566,Z 798.911,A -85,B 0,C 180,E1 -1721.074,E2 -1721.074} C_VEL
LIN {X 0,Y 580.588,Z 785.26,A -85,B 0,C 180,E1 -1721.693,E2 -1721.693} C_VEL
LIN {X 0,Y 580.664,Z 773.797,A -85,B 0,C 180,E1 -1722.068,E2 -1722.068} C_VEL
LIN {X 0,Y 580.732,Z 761.979,A -85,B 0,C 180,E1 -1722.332,E2 -1722.332} C_VEL
LIN {X 0,Y 580.801,Z 682.159,A -85,B 0,C 180,E1 -1723.344,E2 -1723.344} C_VEL
LIN {X 0,Y 580.271,Z 680.201,A -85,B 0,C 180,E1 -1723.388,E2 -1723.388} C_VEL
LIN {X 0,Y 580.254,Z 680.202,A -85,B 0,C 180,E1 -1726.169,E2 -1726.169} C_VEL
LIN {X 0,Y 580.281,Z 680.203,A -85,B 0,C 180,E1 -1729.145,E2 -1729.145} C_VEL
LIN {X 0,Y 580.235,Z 680.202,A -85,B 0,C 180,E1 -1732.048,E2 -1732.048} C_VEL
LIN {X 0,Y 580.262,Z 680.209,A -85,B 0,C 180,E1 -1735.075,E2 -1735.075} C_VEL
LIN {X 0,Y 580.269,Z 680.198,A -85,B 0,C 180,E1 -1737.852,E2 -1737.852} C_VEL
LIN {X 0,Y 580.251,Z 680.202,A -85,B 0,C 180,E1 -1740.688,E2 -1740.688} C_VEL
LIN {X 0,Y 580.269,Z 680.209,A -85,B 0,C 180,E1 -1743.311,E2 -1743.311} C_VEL
LIN {X 0,Y 580.232,Z 680.207,A -85,B 0,C 180,E1 -1745.754,E2 -1745.754} C_VEL
LIN {X 0,Y 580.245,Z 680.2,A -85,B 0,C 180,E1 -1748.141,E2 -1748.141} C_VEL
LIN {X 0,Y 580.274,Z 680.198,A -85,B 0,C 180,E1 -1750.836,E2 -1750.836} C_VEL
LIN {X 0,Y 580.239,Z 680.21,A -85,B 0,C 180,E1 -1753.651,E2 -1753.651} C_VEL
LIN {X 0,Y 580.235,Z 680.201,A -85,B 0,C 180,E1 -1756.603,E2 -1756.603} C_VEL
LIN {X 0,Y 580.273,Z 680.199,A -85,B 0,C 180,E1 -1759.154,E2 -1759.154} C_VEL
LIN {X 0,Y 580.256,Z 680.21,A -85,B 0,C 180,E1 -1761.919,E2 -1761.919} C_VEL
LIN {X 0,Y 580.247,Z 680.203,A -85,B 0,C 180,E1 -1764.452,E2 -1764.452} C_VEL
LIN {X 0,Y 580.234,Z 680.201,A -85,B 0,C 180,E1 -1766.971,E2 -1766.971} C_VEL
LIN {X 0,Y 580.262,Z 680.199,A -85,B 0,C 180,E1 -1769.423,E2 -1769.423} C_VEL
LIN {X 0,Y 580.253,Z 680.209,A -85,B 0,C 180,E1 -1772.132,E2 -1772.132} C_VEL
LIN {X 0,Y 580.254,Z 680.2,A -85,B 0,C 180,E1 -1774.918,E2 -1774.918} C_VEL
LIN {X 0,Y 580.215,Z 680.208,A -85,B 0,C 180,E1 -1777.945,E2 -1777.945} C_VEL
LIN {X 0,Y 580.241,Z 680.203,A -85,B 0,C 180,E1 -1780.911,E2 -1780.911} C_VEL
LIN {X 0,Y 580.252,Z 680.201,A -85,B 0,C 180,E1 -1783.101,E2 -1783.101} C_VEL
LIN {X 0,Y 580.266,Z 680.2,A -85,B 0,C 180,E1 -1785.981,E2 -1785.981} C_VEL
LIN {X 0,Y 580.309,Z 680.2,A -85,B 0,C 180,E1 -1788.827,E2 -1788.827} C_VEL
LIN {X 0,Y 580.263,Z 680.198,A -85,B 0,C 180,E1 -1791.643,E2 -1791.643} C_VEL
LIN {X 0,Y 580.286,Z 680.2,A -85,B 0,C 180,E1 -1794.44,E2 -1794.44} C_VEL
LIN {X 0,Y 580.282,Z 680.202,A -85,B 0,C 180,E1 -1797.223,E2 -1797.223} C_VEL
LIN {X 0,Y 580.268,Z 680.198,A -85,B 0,C 180,E1 -1800,E2 -1800} C_VEL
LIN {X 0,Y 580.282,Z 680.201,A -85,B 0,C 180,E1 -1802.777,E2 -1802.777} C_VEL
LIN {X 0,Y 580.286,Z 680.2,A -85,B 0,C 180,E1 -1805.56,E2 -1805.56} C_VEL
LIN {X 0,Y 580.263,Z 680.198,A -85,B 0,C 180,E1 -1808.357,E2 -1808.357} C_VEL
LIN {X 0,Y 580.302,Z 680.202,A -85,B 0,C 180,E1 -1811.235,E2 -1811.235} C_VEL
LIN {X 0,Y 580.249,Z 680.2,A -85,B 0,C 180,E1 -1814.347,E2 -1814.347} C_VEL
LIN {X 0,Y 580.24,Z 680.203,A -85,B 0,C 180,E1 -1816.919,E2 -1816.919} C_VEL
LIN {X 0,Y 580.245,Z 680.206,A -85,B 0,C 180,E1 -1819.825,E2 -1819.825} C_VEL
LIN {X 0,Y 580.228,Z 680.203,A -85,B 0,C 180,E1 -1822.805,E2 -1822.805} C_VEL
LIN {X 0,Y 580.258,Z 680.2,A -85,B 0,C 180,E1 -1825.082,E2 -1825.082} C_VEL
LIN {X 0,Y 580.253,Z 680.21,A -85,B 0,C 180,E1 -1827.868,E2 -1827.868} C_VEL
LIN {X 0,Y 580.249,Z 680.2,A -85,B 0,C 180,E1 -1830.704,E2 -1830.704} C_VEL
LIN {X 0,Y 580.248,Z 680.201,A -85,B 0,C 180,E1 -1833.322,E2 -1833.322} C_VEL
LIN {X 0,Y 580.268,Z 680.203,A -85,B 0,C 180,E1 -1835.773,E2 -1835.773} C_VEL
LIN {X 0,Y 580.254,Z 680.208,A -85,B 0,C 180,E1 -1838.149,E2 -1838.149} C_VEL
LIN {X 0,Y 580.272,Z 680.199,A -85,B 0,C 180,E1 -1840.846,E2 -1840.846} C_VEL
LIN {X 0,Y 580.24,Z 680.203,A -85,B 0,C 180,E1 -1843.662,E2 -1843.662} C_VEL
LIN {X 0,Y 580.236,Z 680.208,A -85,B 0,C 180,E1 -1846.614,E2 -1846.614} C_VEL
LIN {X 0,Y 580.274,Z 680.198,A -85,B 0,C 180,E1 -1849.164,E2 -1849.164} C_VEL
LIN {X 0,Y 580.247,Z 680.202,A -85,B 0,C 180,E1 -1851.933,E2 -1851.933} C_VEL
LIN {X 0,Y 580.26,Z 680.207,A -85,B 0,C 180,E1 -1854.462,E2 -1854.462} C_VEL
LIN {X 0,Y 580.256,Z 680.206,A -85,B 0,C 180,E1 -1856.981,E2 -1856.981} C_VEL
LIN {X 0,Y 580.259,Z 680.201,A -85,B 0,C 180,E1 -1859.431,E2 -1859.431} C_VEL
LIN {X 0,Y 580.268,Z 680.202,A -85,B 0,C 180,E1 -1862.147,E2 -1862.147} C_VEL
LIN {X 0,Y 580.291,Z 680.351,A -85,B 0,C 180,E1 -1862.898,E2 -1862.898} C_VEL
LIN {X 0,Y 581.617,Z 686.073,A -85,B 0,C 180,E1 -1863.625,E2 -1863.625} C_VEL
LIN {X 0,Y 581.434,Z 709.767,A -85,B 0,C 180,E1 -1866.309,E2 -1866.309} C_VEL
LIN {X 0,Y 581.078,Z 736.661,A -85,B 0,C 180,E1 -1869.288,E2 -1869.288} C_VEL
LIN {X 0,Y 580.829,Z 761.874,A -85,B 0,C 180,E1 -1872.034,E2 -1872.034} C_VEL
LIN {X 0,Y 580.586,Z 787.088,A -85,B 0,C 180,E1 -1874.741,E2 -1874.741} C_VEL
LIN {X 0,Y 580.503,Z 802.141,A -85,B 0,C 180,E1 -1876.32,E2 -1876.32} C_VEL
LIN {X 0,Y 580.938,Z 808.176,A -85,B 0,C 180,E1 -1876.405,E2 -1876.405} C_VEL
LIN {X 0,Y 580.78,Z 912.233,A -85,B 0,C 180,E1 -1877.713,E2 -1877.713} C_VEL
LIN {X 0,Y 580.711,Z 925.404,A -85,B 0,C 180,E1 -1878.022,E2 -1878.022} C_VEL
LIN {X 0,Y 580.623,Z 938.238,A -85,B 0,C 180,E1 -1878.47,E2 -1878.47} C_VEL
LIN {X 0,Y 580.561,Z 949.73,A -85,B 0,C 180,E1 -1879.014,E2 -1879.014} C_VEL
LIN {X 0,Y 580.419,Z 961.279,A -85,B 0,C 180,E1 -1879.717,E2 -1879.717} C_VEL
LIN {X 0,Y 580.39,Z 971.661,A -85,B 0,C 180,E1 -1880.509,E2 -1880.509} C_VEL
LIN {X 0,Y 580.264,Z 980.088,A -85,B 0,C 180,E1 -1881.297,E2 -1881.297} C_VEL
LIN {X 0,Y 580.218,Z 988.003,A -85,B 0,C 180,E1 -1882.173,E2 -1882.173} C_VEL
LIN {X 0,Y 580.153,Z 995.661,A -85,B 0,C 180,E1 -1883.223,E2 -1883.223} C_VEL
LIN {X 0,Y 580.137,Z 1002.706,A -85,B 0,C 180,E1 -1884.443,E2 -1884.443} C_VEL
LIN {X 0,Y 580.107,Z 1007.391,A -85,B 0,C 180,E1 -1885.488,E2 -1885.488} C_VEL
LIN {X 0,Y 580.122,Z 1010.972,A -85,B 0,C 180,E1 -1886.532,E2 -1886.532} C_VEL
LIN {X 0,Y 580.043,Z 1012.821,A -85,B 0,C 180,E1 -1887.227,E2 -1887.227} C_VEL
LIN {X 0,Y 580.038,Z 1014.209,A -85,B 0,C 180,E1 -1887.922,E2 -1887.922} C_VEL
LIN {X 0,Y 580.04,Z 1015.788,A -85,B 0,C 180,E1 -1889.31,E2 -1889.31} C_VEL
LIN {X 0,Y 580.037,Z 1016,A -85,B 0,C 180,E1 -1890.005,E2 -1890.005} C_VEL
LIN {X 0,Y 580.046,Z 1015.18,A -85,B 0,C 180,E1 -1891.393,E2 -1891.393} C_VEL
LIN {X 0,Y 580.038,Z 1014.193,A -85,B 0,C 180,E1 -1892.088,E2 -1892.088} C_VEL
LIN {X 0,Y 580.043,Z 1012.798,A -85,B 0,C 180,E1 -1892.782,E2 -1892.782} C_VEL
LIN {X 0,Y 580.11,Z 1009.882,A -85,B 0,C 180,E1 -1893.825,E2 -1893.825} C_VEL
LIN {X 0,Y 580.054,Z 1005.932,A -85,B 0,C 180,E1 -1894.87,E2 -1894.87} C_VEL
LIN {X 0,Y 580.141,Z 999.853,A -85,B 0,C 180,E1 -1896.089,E2 -1896.089} C_VEL
LIN {X 0,Y 580.188,Z 993.207,A -85,B 0,C 180,E1 -1897.136,E2 -1897.136} C_VEL
LIN {X 0,Y 580.249,Z 984.955,A -85,B 0,C 180,E1 -1898.186,E2 -1898.186} C_VEL
LIN {X 0,Y 580.335,Z 974.556,A -85,B 0,C 180,E1 -1899.238,E2 -1899.238} C_VEL
LIN {X 0,Y 580.438,Z 964.876,A -85,B 0,C 180,E1 -1900.028,E2 -1900.028} C_VEL
LIN {X 0,Y 580.537,Z 954.261,A -85,B 0,C 180,E1 -1900.731,E2 -1900.731} C_VEL
LIN {X 0,Y 580.605,Z 942.575,A -85,B 0,C 180,E1 -1901.34,E2 -1901.34} C_VEL
LIN {X 0,Y 580.662,Z 930.066,A -85,B 0,C 180,E1 -1901.833,E2 -1901.833} C_VEL
LIN {X 0,Y 580.738,Z 917.361,A -85,B 0,C 180,E1 -1902.186,E2 -1902.186} C_VEL
LIN {X 0,Y 580.773,Z 904,A -85,B 0,C 180,E1 -1902.407,E2 -1902.407} C_VEL
LIN {X 0,Y 580.804,Z 804.287,A -85,B 0,C 180,E1 -1903.646,E2 -1903.646} C_VEL
LIN {X 0,Y 580.46,Z 801.706,A -85,B 0,C 180,E1 -1903.705,E2 -1903.705} C_VEL
LIN {X 0,Y 580.695,Z 776.913,A -85,B 0,C 180,E1 -1906.347,E2 -1906.347} C_VEL
LIN {X 0,Y 580.974,Z 747.721,A -85,B 0,C 180,E1 -1909.502,E2 -1909.502} C_VEL
LIN {X 0,Y 581.258,Z 721.444,A -85,B 0,C 180,E1 -1912.391,E2 -1912.391} C_VEL
LIN {X 0,Y 581.572,Z 696.23,A -85,B 0,C 180,E1 -1915.216,E2 -1915.216} C_VEL
LIN {X 0,Y 581.628,Z 686.095,A -85,B 0,C 180,E1 -1916.372,E2 -1916.372} C_VEL
LIN {X 0,Y 580.286,Z 680.207,A -85,B 0,C 180,E1 -1917.137,E2 -1917.137} C_VEL
LIN {X 0,Y 580.236,Z 680.205,A -85,B 0,C 180,E1 -1919.779,E2 -1919.779} C_VEL
LIN {X 0,Y 580.25,Z 680.201,A -85,B 0,C 180,E1 -1922.206,E2 -1922.206} C_VEL
LIN {X 0,Y 580.22,Z 680.209,A -85,B 0,C 180,E1 -1924.704,E2 -1924.704} C_VEL
LIN {X 0,Y 580.258,Z 680.208,A -85,B 0,C 180,E1 -1927.274,E2 -1927.274} C_VEL
LIN {X 0,Y 580.248,Z 680.201,A -85,B 0,C 180,E1 -1930.265,E2 -1930.265} C_VEL
LIN {X 0,Y 580.252,Z 680.203,A -85,B 0,C 180,E1 -1932.711,E2 -1932.711} C_VEL
LIN {X 0,Y 580.258,Z 680.203,A -85,B 0,C 180,E1 -1935.613,E2 -1935.613} C_VEL
LIN {X 0,Y 580.251,Z 680.2,A -85,B 0,C 180,E1 -1938.228,E2 -1938.228} C_VEL
LIN {X 0,Y 580.273,Z 680.203,A -85,B 0,C 180,E1 -1940.964,E2 -1940.964} C_VEL
LIN {X 0,Y 580.253,Z 680.205,A -85,B 0,C 180,E1 -1943.595,E2 -1943.595} C_VEL
LIN {X 0,Y 580.286,Z 680.196,A -85,B 0,C 180,E1 -1946.143,E2 -1946.143} C_VEL
LIN {X 0,Y 580.277,Z 680.198,A -85,B 0,C 180,E1 -1948.614,E2 -1948.614} C_VEL
LIN {X 0,Y 580.296,Z 680.2,A -85,B 0,C 180,E1 -1951.024,E2 -1951.024} C_VEL
LIN {X 0,Y 580.269,Z 680.199,A -85,B 0,C 180,E1 -1954.15,E2 -1954.15} C_VEL
LIN {X 0,Y 580.275,Z 680.198,A -85,B 0,C 180,E1 -1956.442,E2 -1956.442} C_VEL
LIN {X 0,Y 580.279,Z 680.207,A -85,B 0,C 180,E1 -1959.437,E2 -1959.437} C_VEL
LIN {X 0,Y 580.269,Z 680.205,A -85,B 0,C 180,E1 -1961.645,E2 -1961.645} C_VEL
LIN {X 0,Y 580.272,Z 680.203,A -85,B 0,C 180,E1 -1963.825,E2 -1963.825} C_VEL
LIN {X 0,Y 580.307,Z 680.196,A -85,B 0,C 180,E1 -1966.708,E2 -1966.708} C_VEL
LIN {X 0,Y 580.951,Z 682.719,A -85,B 0,C 180,E1 -1966.756,E2 -1966.756} C_VEL
LIN {X 0,Y 580.782,Z 761.792,A -85,B 0,C 180,E1 -1967.752,E2 -1967.752} C_VEL
LIN {X 0,Y 580.744,Z 774.378,A -85,B 0,C 180,E1 -1968.039,E2 -1968.039} C_VEL
LIN {X 0,Y 580.67,Z 787.362,A -85,B 0,C 180,E1 -1968.481,E2 -1968.481} C_VEL
LIN {X 0,Y 580.586,Z 798.785,A -85,B 0,C 180,E1 -1969.009,E2 -1969.009} C_VEL
LIN {X 0,Y 580.413,Z 810.491,A -85,B 0,C 180,E1 -1969.712,E2 -1969.712} C_VEL
LIN {X 0,Y 580.356,Z 819.955,A -85,B 0,C 180,E1 -1970.415,E2 -1970.415} C_VEL
LIN {X 0,Y 580.265,Z 829.616,A -85,B 0,C 180,E1 -1971.292,E2 -1971.292} C_VEL
LIN {X 0,Y 580.223,Z 838.985,A -85,B 0,C 180,E1 -1972.343,E2 -1972.343} C_VEL
LIN {X 0,Y 580.143,Z 846.525,A -85,B 0,C 180,E1 -1973.404,E2 -1973.404} C_VEL
LIN {X 0,Y 580.14,Z 852.426,A -85,B 0,C 180,E1 -1974.438,E2 -1974.438} C_VEL
LIN {X 0,Y 580.108,Z 857.162,A -85,B 0,C 180,E1 -1975.483,E2 -1975.483} C_VEL
LIN {X 0,Y 580.124,Z 860.797,A -85,B 0,C 180,E1 -1976.527,E2 -1976.527} C_VEL
LIN {X 0,Y 580.043,Z 862.684,A -85,B 0,C 180,E1 -1977.222,E2 -1977.222} C_VEL
LIN {X 0,Y 580.038,Z 864.133,A -85,B 0,C 180,E1 -1977.917,E2 -1977.917} C_VEL
LIN {X 0,Y 580.041,Z 865.755,A -85,B 0,C 180,E1 -1979.306,E2 -1979.306} C_VEL
LIN {X 0,Y 580.038,Z 865.996,A -85,B 0,C 180,E1 -1980,E2 -1980} C_VEL
LIN {X 0,Y 580.047,Z 865.231,A -85,B 0,C 180,E1 -1981.389,E2 -1981.389} C_VEL
LIN {X 0,Y 580.038,Z 864.277,A -85,B 0,C 180,E1 -1982.083,E2 -1982.083} C_VEL
LIN {X 0,Y 580.124,Z 861.072,A -85,B 0,C 180,E1 -1983.473,E2 -1983.473} C_VEL
LIN {X 0,Y 580.108,Z 857.525,A -85,B 0,C 180,E1 -1984.517,E2 -1984.517} C_VEL
LIN {X 0,Y 580.138,Z 852.881,A -85,B 0,C 180,E1 -1985.562,E2 -1985.562} C_VEL
LIN {X 0,Y 580.138,Z 847.086,A -85,B 0,C 180,E1 -1986.596,E2 -1986.596} C_VEL
LIN {X 0,Y 580.222,Z 839.683,A -85,B 0,C 180,E1 -1987.657,E2 -1987.657} C_VEL
LIN {X 0,Y 580.255,Z 830.485,A -85,B 0,C 180,E1 -1988.708,E2 -1988.708} C_VEL
LIN {X 0,Y 580.356,Z 821.053,A -85,B 0,C 180,E1 -1989.585,E2 -1989.585} C_VEL
LIN {X 0,Y 580.408,Z 811.809,A -85,B 0,C 180,E1 -1990.289,E2 -1990.289} C_VEL
LIN {X 0,Y 580.543,Z 801.942,A -85,B 0,C 180,E1 -1990.904,E2 -1990.904} C_VEL
LIN {X 0,Y 580.6,Z 791.465,A -85,B 0,C 180,E1 -1991.432,E2 -1991.432} C_VEL
LIN {X 0,Y 580.706,Z 780.17,A -85,B 0,C 180,E1 -1991.873,E2 -1991.873} C_VEL
LIN {X 0,Y 580.76,Z 766.526,A -85,B 0,C 180,E1 -1992.249,E2 -1992.249} C_VEL
LIN {X 0,Y 580.811,Z 752.563,A -85,B 0,C 180,E1 -1992.469,E2 -1992.469} C_VEL
